Q_stMasterDevState.bDcNotInSync 		:=
	(I_nMasterDevState
		AND 16#1000) = 16#1000;

nMasterDevStatePrev 						:=
	I_nMasterDevState;

// ENDE
END_ACTION

ACTION k_SlaveErrorMessage:
	(* CRC-Fehler ------------------------------------------------------------------------- *)
	(* Anzahl der CRC-Fehler am Port A *)
	IF Q_arrDiagSlaveInfo[nIndexSlave].stPortCRCErrors.portA > 0 THEN
			arrFmEcDiagSlaveError[nIndexErrorMessage] :=
				CONCAT(	'Status EtherCAT-Bus: Teilnehmer: ',
							Q_arrDiagSlaveInfo[nIndexSlave].sName);

			arrFmEcDiagSlaveError[nIndexErrorMessage] :=
				CONCAT(	arrFmEcDiagSlaveError[nIndexErrorMessage],
							', Typ: ');

			arrFmEcDiagSlaveError[nIndexErrorMessage] :=
				CONCAT(	arrFmEcDiagSlaveError[nIndexErrorMessage],
							Q_arrDiagSlaveInfo[nIndexSlave].sType);
	
			arrFmEcDiagSlaveError[nIndexErrorMessage] :=
				CONCAT(	arrFmEcDiagSlaveError[nIndexErrorMessage],
							': Anzahl der CRC-Fehler am Port A: ');

			arrFmEcDiagSlaveError[nIndexErrorMessage] :=
				CONCAT(	arrFmEcDiagSlaveError[nIndexErrorMessage],
							UDINT_TO_STRING(Q_arrDiagSlaveInfo[nIndexSlave].stPortCRCErrors.portA));
	END_IF

	(* Anzahl der CRC-Fehler am Port B *)
	IF Q_arrDiagSlaveInfo[nIndexSlave].stPortCRCErrors.portB > 0 THEN
			arrFmEcDiagSlaveError[nIndexErrorMessage] :=
				CONCAT(	'Status EtherCAT-Bus: Teilnehmer: ',
							Q_arrDiagSlaveInfo[nIndexSlave].sName);

			arrFmEcDiagSlaveError[nIndexErrorMessage] :=
				CONCAT(	arrFmEcDiagSlaveError[nIndexErrorMessage],
							', Typ: ');
	
			arrFmEcDiagSlaveError[nIndexErrorMessage] :=
				CONCAT(	arrFmEcDiagSlaveError[nIndexErrorMessage],
							Q_arrDiagSlaveInfo[nIndexSlave].sType);
	
			arrFmEcDiagSlaveError[nIndexErrorMessage] :=
				CONCAT(	arrFmEcDiagSlaveError[nIndexErrorMessage],
							': Anzahl der CRC-Fehler am Port B: ');
	
			arrFmEcDiagSlaveError[nIndexErrorMessage] :=
				CONCAT(	arrFmEcDiagSlaveError[nIndexErrorMessage],
							UDINT_TO_STRING(Q_arrDiagSlaveInfo[nIndexSlave].stPortCRCErrors.portB));
	END_IF

	(* Anzahl der CRC-Fehler am Port C *)
	IF Q_arrDiagSlaveInfo[nIndexSlave].stPortCRCErrors.portC > 0 THEN
			arrFmEcDiagSlaveError[nIndexErrorMessage] :=
				CONCAT(	'Status EtherCAT-Bus: Teilnehmer: ',
							Q_arrDiagSlaveInfo[nIndexSlave].sName);
	
			arrFmEcDiagSlaveError[nIndexErrorMessage] :=
				CONCAT(	arrFmEcDiagSlaveError[nIndexErrorMessage],
							', Typ: ');

			arrFmEcDiagSlaveError[nIndexErrorMessage] :=
				CONCAT(	arrFmEcDiagSlaveError[nIndexErrorMessage],
							Q_arrDiagSlaveInfo[nIndexSlave].sType);
	
			arrFmEcDiagSlaveError[nIndexErrorMessage] :=
				CONCAT(	arrFmEcDiagSlaveError[nIndexErrorMessage],
							': Anzahl der CRC-Fehler am Port C: ');
	
			arrFmEcDiagSlaveError[nIndexErrorMessage] :=
				CONCAT(	arrFmEcDiagSlaveError[nIndexErrorMessage],
							UDINT_TO_STRING(Q_arrDiagSlaveInfo[nIndexSlave].stPortCRCErrors.portC));
	END_IF
	
	(* Anzahl der CRC-Fehler am Port D *)
	IF Q_arrDiagSlaveInfo[nIndexSlave].stPortCRCErrors.portD > 0 THEN
			arrFmEcDiagSlaveError[nIndexErrorMessage] :=
				CONCAT(	'Status EtherCAT-Bus: Teilnehmer: ',
							Q_arrDiagSlaveInfo[nIndexSlave].sName);
	
			arrFmEcDiagSlaveError[nIndexErrorMessage] :=
				CONCAT(	arrFmEcDiagSlaveError[nIndexErrorMessage],
							', Typ: ');
	
			arrFmEcDiagSlaveError[nIndexErrorMessage] :=
				CONCAT(	arrFmEcDiagSlaveError[nIndexErrorMessage],
							Q_arrDiagSlaveInfo[nIndexSlave].sType);
	
			arrFmEcDiagSlaveError[nIndexErrorMessage] :=
				CONCAT(	arrFmEcDiagSlaveError[nIndexErrorMessage],
							': Anzahl der CRC-Fehler am Port D: ');
	
			arrFmEcDiagSlaveError[nIndexErrorMessage] :=
				CONCAT(	arrFmEcDiagSlaveError[nIndexErrorMessage],
							UDINT_TO_STRING(Q_arrDiagSlaveInfo[nIndexSlave].stPortCRCErrors.portD));
	END_IF
	
	(* ------------------------------------------------------------------------------------ *)
	
	(* Link am angegebenen Port fehlt (Port = A, B, C or D) *)
	IF Q_arrDiagSlaveInfo[nIndexSlave].stState.bMissingLink THEN
	
		arrFmEcDiagSlaveError[nIndexErrorMessage] :=
			CONCAT(	'Fehler EtherCAT-Bus: Teilnehmer: ',
						Q_arrDiagSlaveInfo[nIndexSlave].sName);
	
		arrFmEcDiagSlaveError[nIndexErrorMessage] :=
			CONCAT(	arrFmEcDiagSlaveError[nIndexErrorMessage],
						', Typ: ');
	
		arrFmEcDiagSlaveError[nIndexErrorMessage] :=
			CONCAT(	arrFmEcDiagSlaveError[nIndexErrorMessage],
						Q_arrDiagSlaveInfo[nIndexSlave].sType);
	
		IF Q_arrDiagSlaveInfo[nIndexSlave].stState.bPortA THEN
			arrFmEcDiagSlaveError[nIndexErrorMessage] :=
					CONCAT(	arrFmEcDiagSlaveError[nIndexErrorMessage],
								': Link am Port A fehlt !');
		ELSIF Q_arrDiagSlaveInfo[nIndexSlave].stState.bPortB THEN
			arrFmEcDiagSlaveError[nIndexErrorMessage] :=
				CONCAT(	arrFmEcDiagSlaveError[nIndexErrorMessage],
							': Link am Port B fehlt !');
		ELSIF Q_arrDiagSlaveInfo[nIndexSlave].stState.bPortC THEN
			arrFmEcDiagSlaveError[nIndexErrorMessage] :=
				CONCAT(	arrFmEcDiagSlaveError[nIndexErrorMessage],
							': Link am Port C fehlt !');
		ELSIF Q_arrDiagSlaveInfo[nIndexSlave].stState.bPortD THEN
			arrFmEcDiagSlaveError[nIndexErrorMessage] :=
				CONCAT(	arrFmEcDiagSlaveError[nIndexErrorMessage],
							': Link am Port D fehlt !');
		END_IF
	
		IF nIndexErrorMessage < cMaxAnzahlSlaveError THEN
			nIndexErrorMessage := nIndexErrorMessage + 1;
		ELSE
			RETURN;
		END_IF

	(* Ein zusätzlicher Link wurde am angegebenen Port festgestellt *)
	ELSIF Q_arrDiagSlaveInfo[nIndexSlave].stState.bUnexpectedLink THEN
	
		arrFmEcDiagSlaveError[nIndexErrorMessage] :=
			CONCAT(	'Fehler EtherCAT-Bus: Teilnehmer: ',
						Q_arrDiagSlaveInfo[nIndexSlave].sName);
	
		arrFmEcDiagSlaveError[nIndexErrorMessage] :=
			CONCAT(	arrFmEcDiagSlaveError[nIndexErrorMessage],
						', Typ: ');
	
		arrFmEcDiagSlaveError[nIndexErrorMessage] :=
			CONCAT(	arrFmEcDiagSlaveError[nIndexErrorMessage],
						Q_arrDiagSlaveInfo[nIndexSlave].sType);
	
		IF Q_arrDiagSlaveInfo[nIndexSlave].stState.bPortA THEN
			arrFmEcDiagSlaveError[nIndexErrorMessage] :=
					CONCAT(	arrFmEcDiagSlaveError[nIndexErrorMessage],
								': Ein zusätzlicher Link wurde am Port A festgestellt !');
		ELSIF Q_arrDiagSlaveInfo[nIndexSlave].stState.bPortB THEN
			arrFmEcDiagSlaveError[nIndexErrorMessage] :=
				CONCAT(	arrFmEcDiagSlaveError[nIndexErrorMessage],
								': Ein zusätzlicher Link wurde am Port B festgestellt !');
		ELSIF Q_arrDiagSlaveInfo[nIndexSlave].stState.bPortC THEN
			arrFmEcDiagSlaveError[nIndexErrorMessage] :=
				CONCAT(	arrFmEcDiagSlaveError[nIndexErrorMessage],
								': Ein zusätzlicher Link wurde am Port C festgestellt !');
		ELSIF Q_arrDiagSlaveInfo[nIndexSlave].stState.bPortD THEN
			arrFmEcDiagSlaveError[nIndexErrorMessage] :=
				CONCAT(	arrFmEcDiagSlaveError[nIndexErrorMessage],
								': Ein zusätzlicher Link wurde am Port D festgestellt !');
		END_IF
	
		IF nIndexErrorMessage < cMaxAnzahlSlaveError THEN
			nIndexErrorMessage := nIndexErrorMessage + 1;
		ELSE
			RETURN;
		END_IF

	(* Ein Link ohne Kommunikation wurde festgestellt *)
	ELSIF Q_arrDiagSlaveInfo[nIndexSlave].stState.bLinkError THEN
	
		arrFmEcDiagSlaveError[nIndexErrorMessage] :=
			CONCAT(	'Fehler EtherCAT-Bus: Teilnehmer: ',
						Q_arrDiagSlaveInfo[nIndexSlave].sName);
	
		arrFmEcDiagSlaveError[nIndexErrorMessage] :=
			CONCAT(	arrFmEcDiagSlaveError[nIndexErrorMessage],
						', Typ: ');
	
		arrFmEcDiagSlaveError[nIndexErrorMessage] :=
			CONCAT(	arrFmEcDiagSlaveError[nIndexErrorMessage],
						Q_arrDiagSlaveInfo[nIndexSlave].sType);
	
		IF Q_arrDiagSlaveInfo[nIndexSlave].stState.bPortA THEN
			arrFmEcDiagSlaveError[nIndexErrorMessage] :=
					CONCAT(	arrFmEcDiagSlaveError[nIndexErrorMessage],
								': Am Port A wurde ein Link ohne Kommunikation festgestellt !');
		ELSIF Q_arrDiagSlaveInfo[nIndexSlave].stState.bPortB THEN
			arrFmEcDiagSlaveError[nIndexErrorMessage] :=
				CONCAT(	arrFmEcDiagSlaveError[nIndexErrorMessage],
								': Am Port B wurde ein Link ohne Kommunikation festgestellt !');
		ELSIF Q_arrDiagSlaveInfo[nIndexSlave].stState.bPortC THEN
			arrFmEcDiagSlaveError[nIndexErrorMessage] :=
				CONCAT(	arrFmEcDiagSlaveError[nIndexErrorMessage],
								': Am Port C wurde ein Link ohne Kommunikation festgestellt !');
		ELSIF Q_arrDiagSlaveInfo[nIndexSlave].stState.bPortD THEN
			arrFmEcDiagSlaveError[nIndexErrorMessage] :=
				CONCAT(	arrFmEcDiagSlaveError[nIndexErrorMessage],
								': Am Port D wurde ein Link ohne Kommunikation festgestellt !');
		END_IF
	
		IF nIndexErrorMessage < cMaxAnzahlSlaveError THEN
			nIndexErrorMessage := nIndexErrorMessage + 1;
		ELSE
			RETURN;
		END_IF
	
	END_IF

	
	(* Fehler Slave nicht erkannt *)
	IF Q_arrDiagSlaveInfo[nIndexSlave].stState.bNoCommToSlave THEN
	
		arrFmEcDiagSlaveError[nIndexErrorMessage] :=
			CONCAT(	'Fehler EtherCAT-Bus: Teilnehmer: ',
						Q_arrDiagSlaveInfo[nIndexSlave].sName);
	
		arrFmEcDiagSlaveError[nIndexErrorMessage] :=
			CONCAT(	arrFmEcDiagSlaveError[nIndexErrorMessage],
						', Typ: ');
	
		arrFmEcDiagSlaveError[nIndexErrorMessage] :=
			CONCAT(	arrFmEcDiagSlaveError[nIndexErrorMessage],
						Q_arrDiagSlaveInfo[nIndexSlave].sType);

		arrFmEcDiagSlaveError[nIndexErrorMessage] :=
			CONCAT(	arrFmEcDiagSlaveError[nIndexErrorMessage],
						': State: ');
	
		CASE Q_arrDiagSlaveInfo[nIndexSlave].stState.eEcState OF
	
		eEcState_UNDEFINED:	arrFmEcDiagSlaveError[nIndexErrorMessage] :=
										CONCAT(	arrFmEcDiagSlaveError[nIndexErrorMessage],
													'UNDEFINED');
		eEcState_INIT:			arrFmEcDiagSlaveError[nIndexErrorMessage] :=
										CONCAT(	arrFmEcDiagSlaveError[nIndexErrorMessage],
													'INIT / NO COMMUNICATION');
		eEcState_PREOP:		arrFmEcDiagSlaveError[nIndexErrorMessage] :=
										CONCAT(	arrFmEcDiagSlaveError[nIndexErrorMessage],
													'PREOP');
		eEcState_BOOT:			arrFmEcDiagSlaveError[nIndexErrorMessage] :=
										CONCAT(	arrFmEcDiagSlaveError[nIndexErrorMessage],
													'BOOT');
		eEcState_SAFEOP:		arrFmEcDiagSlaveError[nIndexErrorMessage] :=
										CONCAT(	arrFmEcDiagSlaveError[nIndexErrorMessage],
													'SAFEOP');
		eEcState_OP:			arrFmEcDiagSlaveError[nIndexErrorMessage] :=
										CONCAT(	arrFmEcDiagSlaveError[nIndexErrorMessage],
													'OP');
		END_CASE
	
		IF nIndexErrorMessage < cMaxAnzahlSlaveError THEN
			nIndexErrorMessage := nIndexErrorMessage + 1;
		ELSE
			RETURN;
		END_IF
	END_IF
	
	(* B E *)
END_ACTION

END_FUNCTION_BLOCK

// POUs/EtherCATDiagnose/FB_EtherCATFrameDiag
FUNCTION_BLOCK FB_EtherCATFrameDiag
VAR_INPUT
	I_nFrameXWcState 		: WORD;
	I_nFrameState			: WORD;
END_VAR
VAR_OUTPUT
	Q_bFrameWcStateOK		: BOOL;
	Q_bFrameStateOK		: BOOL;
END_VAR

// set/clear frame flag
Q_bFrameWcStateOK := ((I_nFrameXWcState AND 16#FFFF) = 0);

Q_bFrameStateOK	:= ((I_nFrameState AND 16#FFFF) = 0);

END_FUNCTION_BLOCK

// POUs/EtherCATDiagnose/FB_IoLinkFehler
(*
Date				| Version		| created under			| Author				| Remark 
---------------------------------------------------------------------------------------- 
03/10/2017		| 1.0.0			| V2.11.2258				| H.Gennet			| first release 
*)
(*Pro Zyklus nur einen der 4 Channels, nacheinander.*)
FUNCTION_BLOCK FB_IoLinkFehler
VAR
	// Baustein zum Zusammenfügen von Texten in ein String
	fbFormat 	: Tc2_Utilities.FB_FormatString;

	// Zähler
	nCounter 	: INT; 				(*Zähler für das nState Array*)
	nChannel		: INT;				(*Zähler + 1*)

	// Zwischenspeicher der Input Stati zur besseren Auswertung
	nState 		: ARRAY [0..3] OF USINT;
	
	arrLetzteFehlermeldung	: ARRAY [0..3] OF Tc2_System.T_MaxString;
	arrVerzMeld					: ARRAY [0..3] OF TON;

END_VAR
VAR_IN_OUT
	IQ_stMeldung	: ST_MeldIOLinkKlemme;
END_VAR

VAR_INPUT
	(*BMK Input händisch als String*)
	I_sBMK : 	Tc2_System.T_MaxString;

	(*Input der einzelnen Stati*)
	I_nStateCh1	: USINT;
	I_nStateCh2	: USINT;
	I_nStateCh3	: USINT;
	I_nStateCh4	: USINT;
END_VAR

VAR_OUTPUT
	Q_arrFehlermeldung : ARRAY [0..3] OF Tc2_System.T_MaxString;	// Output der Fehlermeldungen als String-Array
END_VAR

(*Übertragung der einzelnen Stati in ein Array*)
nState[0] := I_nStateCh1;
nState[1] := I_nStateCh2;
nState[2] := I_nStateCh3;
nState[3] := I_nStateCh4;

(*Zurücksetzen des Counters, wenn dieser größer als 3 ist*)
IF nCounter > 3 THEN
	nCounter := 0;
END_IF

nChannel := nCounter +1;
(*Abfrage der aktuellen Stati*)
CASE nState[nCounter] OF
	(*16#00:
		(*Port diasbled*)
		fbFormat(sFormat := '%s Ch %d: Kein Teilnehmer an Ch %d  angeschlossen!',arg1:=F_STRING(sBMK), arg2:=F_INT(nChannel), sOut => sFehlermeldung[nCounter]);
	16#01:
		(*Port in std dig in*)
		fbFormat(sFormat := '%s Ch %d: ist als Standard Input definiert!',arg1:=F_STRING(sBMK), arg2:=F_INT(nChannel), sOut => sFehlermeldung[nCounter]);
	16#02:
		(*Port in std dig out*)
		fbFormat(sFormat := '%s Ch %d: ist als Standard Output definiert!',arg1:=F_STRING(sBMK), arg2:=F_INT(nChannel), sOut => sFehlermeldung[nCounter]);
	16#03:
		(*Port in communikation OP*)
		fbFormat(sFormat := '%s Ch %d: befindet sich im Status OP!',arg1:=F_STRING(sBMK), arg2:=F_INT(nChannel), sOut => sFehlermeldung[nCounter]);*)
	16#04:
		(*Port in communikation Comport*)
		fbFormat(sFormat := '%s Ch %d: Port in communikation Comport!',arg1:=F_STRING(I_sBMK), arg2:=F_INT(nChannel), sOut => Q_arrFehlermeldung[nCounter]);
	16#0B:
		(*Teilnehmer befindet sich im Teach-in Modus*)
		fbFormat(sFormat := '%s Ch %d: eingeteacht!',arg1:=F_STRING(I_sBMK), arg2:=F_INT(nChannel), sOut => Q_arrFehlermeldung[nCounter]);
	16#10:
		(*Watchdog detected*)
		fbFormat(sFormat := '%s Ch %d: Watchdog hat ausgelöst!',arg1:=F_STRING(I_sBMK), arg2:=F_INT(nChannel), sOut => Q_arrFehlermeldung[nCounter]);
	16#20:
		(*internal Error*)
		fbFormat(sFormat := '%s Ch %d: Es gibt einen internen Fehler!',arg1:=F_STRING(I_sBMK), arg2:=F_INT(nChannel), sOut => Q_arrFehlermeldung[nCounter]);
	16#30,16#B0: (*Bei einer falschen Device ID (DeviceDescription) springt der Status zwischen 16#30 und 16#B0*)
		(*invalid Device ID*)
		fbFormat(sFormat := '%s Ch %d: Die Device ID ist fehlerhaft!',arg1:=F_STRING(I_sBMK), arg2:=F_INT(nChannel), sOut => Q_arrFehlermeldung[nCounter]); (* Bitte die korrekte Device Describtion einlesen und den korrekten Teilnehmer auswählen*)
	16#40:
		(*invalid Vendor ID*)
		fbFormat(sFormat := '%s Ch %d: Die Vendor ID ist fehlerhaft!',arg1:=F_STRING(I_sBMK), arg2:=F_INT(nChannel), sOut => Q_arrFehlermeldung[nCounter]);	(* Bitte in der Device Describtion korrigieren. Die Vendor IDs können über Io-Link.com abgerufen werden *)
	16#50:
		(*invalid IO-Link Error*)
		fbFormat(sFormat := '%s Ch %d: Es liegt ein IO-Link Error vor!',arg1:=F_STRING(I_sBMK), arg2:=F_INT(nChannel), sOut => Q_arrFehlermeldung[nCounter]);
	16#60:
		(*invalid Frame Capability*)
		fbFormat(sFormat := '%s Ch %d: Der aktuelle Frame ist ungültig!',arg1:=F_STRING(I_sBMK), arg2:=F_INT(nChannel), sOut => Q_arrFehlermeldung[nCounter]);
	16#70:
		(*invalid Cycle Time*)
		fbFormat(sFormat := '%s Ch %d: Die Zylkuszeit ist ungültig. Bitte die Einstellungen überprüfen!',arg1:=F_STRING(I_sBMK), arg2:=F_INT(nChannel), sOut => Q_arrFehlermeldung[nCounter]);
	16#80:
		(*invalid PD in length*)
		fbFormat(sFormat := '%s Ch %d: Die Länge der eingehenden Prozessdaten passt nicht mit der erwarteten Länge zusammen!',arg1:=F_STRING(I_sBMK), arg2:=F_INT(nChannel), sOut => Q_arrFehlermeldung[nCounter]);
	16#90:
		(*invalid PD out length*)
		fbFormat(sFormat := '%s Ch %d: Die Länge der ausgehenden Prozessdaten passt nicht mit der erwarteten Länge zusammen!',arg1:=F_STRING(I_sBMK), arg2:=F_INT(nChannel), sOut => Q_arrFehlermeldung[nCounter]);
	16#A0:
		(*no Device detected*)
		fbFormat(sFormat := '%s Ch %d: Der Teilnehmer hat den Kontakt verloren!',arg1:=F_STRING(I_sBMK), arg2:=F_INT(nChannel), sOut => Q_arrFehlermeldung[nCounter]); (* Bitte die Anschlüsse und Verbindungskabel prüfen. Wenn dort nichts vorliegt kann der Teilnehmer defekt sein*)
	ELSE
		IF (nState[nCounter] > 16#03) THEN
			(*Unbekannter Zustand, der nicht im Infosys definiert ist*)
			fbFormat(sFormat := '%s Ch %d: Unbekannter Status!',arg1:=F_STRING(I_sBMK), arg2:=F_INT(nChannel), sOut => Q_arrFehlermeldung[nCounter]);
		ELSE
			Q_arrFehlermeldung[nCounter] := '';
		END_IF
END_CASE

nCounter := nCounter+1;

// Zuweisung der Meldungen
IQ_stMeldung.SourceName	:= I_sBMK;

arrVerzMeld[0](
	IN := Q_arrFehlermeldung[0] <> ''
				AND Q_arrFehlermeldung[0] = arrLetzteFehlermeldung[0],
	PT := t#500MS
);

arrVerzMeld[1](
	IN := Q_arrFehlermeldung[1] <> ''
				AND Q_arrFehlermeldung[1] = arrLetzteFehlermeldung[1],
	PT := t#500MS
);

arrVerzMeld[2](
	IN := Q_arrFehlermeldung[2] <> ''
				AND Q_arrFehlermeldung[2] = arrLetzteFehlermeldung[2],
	PT := t#500MS
);

arrVerzMeld[3](
	IN := Q_arrFehlermeldung[3] <> ''
				AND Q_arrFehlermeldung[3] = arrLetzteFehlermeldung[3],
	PT := t#500MS
);

IQ_stMeldung.bMeld1	:= arrVerzMeld[0].Q;
IQ_stMeldung.bMeld2	:= arrVerzMeld[1].Q;
IQ_stMeldung.bMeld3	:= arrVerzMeld[2].Q;
IQ_stMeldung.bMeld4	:= arrVerzMeld[3].Q;
IQ_stMeldung.sText1	:= Q_arrFehlermeldung[0];
IQ_stMeldung.sText2	:= Q_arrFehlermeldung[1];
IQ_stMeldung.sText3	:= Q_arrFehlermeldung[2];
IQ_stMeldung.sText4	:= Q_arrFehlermeldung[3];


arrLetzteFehlermeldung[0] :=  Q_arrFehlermeldung[0];
arrLetzteFehlermeldung[1] :=  Q_arrFehlermeldung[1];
arrLetzteFehlermeldung[2] :=  Q_arrFehlermeldung[2];
arrLetzteFehlermeldung[3] :=  Q_arrFehlermeldung[3];

// ENDE

END_FUNCTION_BLOCK

// POUs/Grundstellung/FB_UniGrdstlgAbl
// Dieser Grundstellungsablauf besteht aus einer Schrittkette mit insgesamt 9 einzelnen Schritten.
// Gesteuert wird er über zwei HMI-Schnittstellen und weiteren Eingängen zum Starten der Grundstellung
FUNCTION_BLOCK FB_UniGrdstlgAbl
VAR_INPUT

	I_sStatName			:Tc2_System.T_MaxString;	// Aktueller Stationsname für Fehlermeldungen

	I_bHandbetrAktiv	:BOOL;	// Betriebsart, Schutzbereich etc.
	I_bGrdstAnwahlFrg	:BOOL;	// Betriebsart, Schutzbereich etc.

	I_bLoeschDatenPos :BOOL;	// Grundstellungsablauf-Anwahl durch Datensatz löschen in der Teileverfolgung
	I_bGrdstlgAnwTast :BOOL;	// Grundstellungsablauf-Anwahl durch Paneltaste, Softkey etc.
	I_bGrdstlgAnfStat	:BOOL;	// Grundstellungsablauf-Anwahl durch extern z.B. Referenzablauf. Bei fallender Flanke wird die Grundstellung wieder abgewählt, bzw. umgeschaltet
	
	I_bDatenVorh		:BOOL;	// Sind Daten vorhanden wird das Lösch-Bit gesetzt
	I_bSensPosFreiErk	:BOOL:= TRUE;	// Optional: Erkennung Teileentnahme. Grundstellung ist erst zuende, wenn dieses Bit TRUE ist.
	I_bTeileEntnahmeNoetig	: BOOL;	// Nur für eine Melden, dass nach der erfolgreichen Grundstellungsfahrt das Teil entnommen werden soll. Die Meldung bleibt so lange an wie die Grundstellung aktiv ist oder dieses Bit gesetzt
	 
	I_bGrdstStep1End	:BOOL:= TRUE;	// Rückmeldung Schritt 1 fertig
	I_bGrdstStep2End	:BOOL:= TRUE;	// Rückmeldung Schritt 2 fertig
	I_bGrdstStep3End	:BOOL:= TRUE;	// Rückmeldung Schritt 3 fertig
	I_bGrdstStep4End	:BOOL:= TRUE;	// Rückmeldung Schritt 4 fertig
	I_bGrdstStep5End	:BOOL:= TRUE;	// Rückmeldung Schritt 5 fertig
	I_bGrdstStep6End	:BOOL:= TRUE;	// Rückmeldung Schritt 6 fertig
	I_bGrdstStep7End	:BOOL:= TRUE;	// Rückmeldung Schritt 7 fertig
	I_bGrdstStep8End	:BOOL:= TRUE;	// Rückmeldung Schritt 8 fertig
	I_bGrdstStep9End	:BOOL:= TRUE;	// Rückmeldung Schritt 9 fertig

	I_bParamEinzelschritte	: BOOL;	// Wenn dieser Parameter an ist, dann sind die Schritte nur einzeln an. Also wenn Q_bGrdstStep2Akt an geht, geht Q_bGrdstStep1Akt aus.
END_VAR
VAR_IN_OUT

	IQ_stUniAnstgEinzelHMI	:ST_UniGrdstlgAbl;	// HMI-Struktur Einzelposition
	IQ_stUniAnstgGesamtHMI	:ST_UniGrdstlgAbl;	// HMI-Struktur Anlagenbereich/Gesamtanlage, Liste mit allen Grundstellungsabläufen

END_VAR
VAR_OUTPUT

	Q_bGrdstAblAktiv	:BOOL;	// Gesamtablauf Aktiv
	Q_bGrdstAblReset	:BOOL;	// Gesamtablauf 1x Reset
	Q_bGrdstAblEnde	:BOOL;	// Gesamtablauf Ausgeführt
	
	Q_bDatenLoeschen	:BOOL;	// Ein vorhandener Datensatz soll gelöscht werden
	 
	Q_bGrdstStep1Akt	:BOOL;	// Ist TRUE sobald die Grundstellung aktiv ist. Wenn der Parameter I_bParamEinzelschritte aktiv ist, dann wirds FALSE wenn der nächste Schritt aktiv ist.
	Q_bGrdstStep2Akt	:BOOL;	// Ist TRUE sobald die Weiterschaltbedingung vom vorherigen TRUE ist. Wenn der Parameter I_bParamEinzelschritte aktiv ist, dann wirds FALSE wenn der nächste Schritt aktiv ist.
	Q_bGrdstStep3Akt	:BOOL;	// Ist TRUE sobald die Weiterschaltbedingung vom vorherigen TRUE ist. Wenn der Parameter I_bParamEinzelschritte aktiv ist, dann wirds FALSE wenn der nächste Schritt aktiv ist.
	Q_bGrdstStep4Akt	:BOOL;	// Ist TRUE sobald die Weiterschaltbedingung vom vorherigen TRUE ist. Wenn der Parameter I_bParamEinzelschritte aktiv ist, dann wirds FALSE wenn der nächste Schritt aktiv ist.
	Q_bGrdstStep5Akt	:BOOL;	// Ist TRUE sobald die Weiterschaltbedingung vom vorherigen TRUE ist. Wenn der Parameter I_bParamEinzelschritte aktiv ist, dann wirds FALSE wenn der nächste Schritt aktiv ist.
	Q_bGrdstStep6Akt	:BOOL;	// Ist TRUE sobald die Weiterschaltbedingung vom vorherigen TRUE ist. Wenn der Parameter I_bParamEinzelschritte aktiv ist, dann wirds FALSE wenn der nächste Schritt aktiv ist.
	Q_bGrdstStep7Akt	:BOOL;	// Ist TRUE sobald die Weiterschaltbedingung vom vorherigen TRUE ist. Wenn der Parameter I_bParamEinzelschritte aktiv ist, dann wirds FALSE wenn der nächste Schritt aktiv ist.
	Q_bGrdstStep8Akt	:BOOL;	// Ist TRUE sobald die Weiterschaltbedingung vom vorherigen TRUE ist. Wenn der Parameter I_bParamEinzelschritte aktiv ist, dann wirds FALSE wenn der nächste Schritt aktiv ist.
	Q_bGrdstStep9Akt	:BOOL;	// Ist TRUE sobald die Weiterschaltbedingung vom vorherigen TRUE ist. Dieser Schritt bleibt solange TRUE wie die Grundstellung aktiv ist.

	Q_bGrdstlgMeldg	:BOOL;	// Grundstellung-Meldung für Paneltaste, Softkey etc. mit Blinktakt wenn aktiv. Durchgehen TRUE, wenn Grundstellung Ende
END_VAR
VAR

	rtrigImpAnAbw		:R_TRIG;
	rtrigDatenLoeschen:R_TRIG;
	bGrdst1xAngw		:BOOL;

	nStepState			:INT;
END_VAR

	(*Uni.- Grundstellungsablauf*)
	
	(**************************************************)	
	(*Grundstellung An.-Abwahl*)

	a_AnAbwahl();
	
	(**************************************************)	
	(*Grundstellung Step-Ablauf*)

	b_StepAblauf();

	(**************************************************)	
	(*Zustände anzeigen*)

	y_ZustAnzg();

	(**************************************************)	
	(*Meldungen ausgeben*)

	z_HinwMeld();
	
	(**************************************************)

ACTION a_AnAbwahl:
	
//****************************************************************************************************
// Grundstellung An.-Abwahl
	
	rtrigDatenLoeschen(CLK:= I_bLoeschDatenPos);
									  
	rtrigImpAnAbw (CLK:= (IQ_stUniAnstgEinzelHMI.stHandFktHMI[1].bySwitch > 0
								OR IQ_stUniAnstgGesamtHMI.stHandFktHMI[1].bySwitch > 0
								OR I_bGrdstlgAnwTast
								OR (I_bGrdstlgAnfStat
									 AND NOT bGrdst1xAngw) 
								OR (NOT I_bGrdstlgAnfStat
									 AND bGrdst1xAngw))
								AND (I_bGrdstAnwahlFrg
									 AND I_bHandbetrAktiv));

//****************************************************************************************************
//ToDo teilweise nur Anwahl /direkter zugriff auf Teileverfolgung...

	Q_bGrdstAblReset:= FALSE;
	
	IF NOT I_bHandbetrAktiv
		THEN
			Q_bGrdstAblAktiv:= FALSE;
			bGrdst1xAngw	 := FALSE;	
			nStepState		 := 0;			
	ELSIF rtrigImpAnAbw.Q
		THEN
			Q_bGrdstAblAktiv:= NOT Q_bGrdstAblAktiv;
			Q_bGrdstAblReset:= Q_bGrdstAblAktiv;
			bGrdst1xAngw	 := I_bGrdstlgAnfStat; //ToDo
			nStepState		 := 0;
			
	ELSIF rtrigDatenLoeschen.Q
		OR (I_bLoeschDatenPos
			AND NOT Q_bGrdstAblAktiv)
		THEN
			Q_bGrdstAblAktiv	:= TRUE;
			Q_bGrdstAblReset:= Q_bGrdstAblAktiv;
			nStepState		 := 0;
	END_IF

//****************************************************************************************************
//
END_ACTION

ACTION b_StepAblauf:
	
//****************************************************************************************************
// Grundstellung Step-Ablauf

	CASE nStepState OF
0:	//Initialisierung

	Q_bDatenLoeschen:=	
	Q_bGrdstStep1Akt:=
	Q_bGrdstStep2Akt:=
	Q_bGrdstStep3Akt:=
	Q_bGrdstStep4Akt:=
	Q_bGrdstStep5Akt:=
	Q_bGrdstStep6Akt:=
	Q_bGrdstStep7Akt:=
	Q_bGrdstStep8Akt:=
	Q_bGrdstStep9Akt:= FALSE;

	IF Q_bGrdstAblAktiv THEN
		nStepState:= 1;
	END_IF
	
1:	//Ablauf Step 1
	Q_bGrdstStep1Akt:= TRUE;
	
	IF I_bGrdstStep1End THEN
		nStepState:= 2;
		Q_bGrdstStep1Akt	:= NOT I_bParamEinzelschritte;
	END_IF
	
2:	//Ablauf Step 2
	Q_bGrdstStep2Akt:= TRUE;
	
	IF I_bGrdstStep2End THEN
		nStepState:= 3;
		Q_bGrdstStep2Akt	:= NOT I_bParamEinzelschritte;
	END_IF
	
3:	//Ablauf Step 3
	Q_bGrdstStep3Akt:= TRUE;
	
	IF I_bGrdstStep3End THEN
		nStepState:= 4;
		Q_bGrdstStep3Akt	:= NOT I_bParamEinzelschritte;
	END_IF
	
4:	//Ablauf Step 4
	Q_bGrdstStep4Akt:= TRUE;
	
	IF I_bGrdstStep4End THEN
		nStepState:= 5;
		Q_bGrdstStep4Akt	:= NOT I_bParamEinzelschritte;
	END_IF
	
5:	//Ablauf Step 5
	Q_bGrdstStep5Akt:= TRUE;
	
	IF I_bGrdstStep5End THEN
		nStepState:= 6;
		Q_bGrdstStep5Akt	:= NOT I_bParamEinzelschritte;
	END_IF
	
6:	//Ablauf Step 6
	Q_bGrdstStep6Akt:= TRUE;
	
	IF I_bGrdstStep6End THEN
		nStepState:= 7;
		Q_bGrdstStep6Akt	:= NOT I_bParamEinzelschritte;
	END_IF
	
7:	//Ablauf Step 7
	Q_bGrdstStep7Akt:= TRUE;
	
	IF I_bGrdstStep7End THEN
		nStepState:= 8;
		Q_bGrdstStep7Akt	:= NOT I_bParamEinzelschritte;
	END_IF
	
8:	//Ablauf Step 8
	Q_bGrdstStep8Akt:= TRUE;
	
	IF I_bGrdstStep8End THEN
		nStepState:= 9;
		Q_bGrdstStep8Akt	:= NOT I_bParamEinzelschritte;
	END_IF
	
9:	//Ablauf Step 9
	Q_bGrdstStep9Akt:= TRUE;
	
	IF I_bGrdstStep9End THEN
		nStepState:= 10;
	END_IF
	
10://Datenabfrage, wenn Daten zum löschen vorhanden sind, bleibt das Lösch-Bit an
	
	IF I_bDatenVorh
		THEN
			Q_bDatenLoeschen	:= TRUE;	
		ELSE
			Q_bDatenLoeschen	:= FALSE;
			nStepState:= 99;
   END_IF

99://Ablaufende	

	END_CASE	

//****************************************************************************************************

	Q_bGrdstAblEnde:= nStepState = 99
							AND I_bSensPosFreiErk;
 
//****************************************************************************************************
END_ACTION

ACTION y_ZustAnzg:

//****************************************************************************************************
// Zustände anzeigen

	IF I_bGrdstAnwahlFrg
		AND I_bHandbetrAktiv
	THEN	// Funktion freigegeben
			IQ_stUniAnstgEinzelHMI.stHandFktHMI[1].sColour	:= cDefaultAsString;
			IQ_stUniAnstgEinzelHMI.stHandFktHMI[1].sText		:= 'ausführen';
			IQ_stUniAnstgGesamtHMI.stHandFktHMI[1].sColour	:= cDefaultAsString;
			IQ_stUniAnstgGesamtHMI.stHandFktHMI[1].sText		:= 'ausführen';
			IQ_stUniAnstgEinzelHMI.stHandFktHMI[1].byStatus	:= 0;
			IQ_stUniAnstgGesamtHMI.stHandFktHMI[1].byStatus	:= 0;
			IQ_stUniAnstgEinzelHMI.stHandFktHMI[1].iDisplayMode	:= 0;
			IQ_stUniAnstgGesamtHMI.stHandFktHMI[1].iDisplayMode	:= 0;

		IF Q_bGrdstAblAktiv
			AND NOT Q_bGrdstAblEnde
		THEN	// Handfunktion aktiv
			IQ_stUniAnstgEinzelHMI.stHandFktHMI[1].sColour	:= cGelbAsString;
			IQ_stUniAnstgEinzelHMI.stHandFktHMI[1].sText		:= 'ausführen';
			IQ_stUniAnstgGesamtHMI.stHandFktHMI[1].sColour	:= cGelbAsString;
			IQ_stUniAnstgGesamtHMI.stHandFktHMI[1].sText		:= 'ausführen';
			IQ_stUniAnstgEinzelHMI.stHandFktHMI[1].byStatus	:= 0;
			IQ_stUniAnstgGesamtHMI.stHandFktHMI[1].byStatus	:= 0;
			IQ_stUniAnstgEinzelHMI.stHandFktHMI[1].iDisplayMode	:= 2;
			IQ_stUniAnstgGesamtHMI.stHandFktHMI[1].iDisplayMode	:= 2;
		END_IF
		
		IF Q_bGrdstAblEnde
		THEN	// Handfunktion ausgeführt
			IQ_stUniAnstgEinzelHMI.stHandFktHMI[1].sColour:= cGruenAsString;
			IQ_stUniAnstgEinzelHMI.stHandFktHMI[1].sText:= 'ausgeführt';
			IQ_stUniAnstgGesamtHMI.stHandFktHMI[1].sColour:= cGruenAsString;
			IQ_stUniAnstgGesamtHMI.stHandFktHMI[1].sText:= 'ausgeführt';
			IQ_stUniAnstgEinzelHMI.stHandFktHMI[1].byStatus:= 0;
			IQ_stUniAnstgGesamtHMI.stHandFktHMI[1].byStatus:= 0;
			IQ_stUniAnstgEinzelHMI.stHandFktHMI[1].iDisplayMode	:= 0;
			IQ_stUniAnstgGesamtHMI.stHandFktHMI[1].iDisplayMode	:= 0;
		END_IF
		
	ELSE	// Funktion gesperrt
		IQ_stUniAnstgEinzelHMI.stHandFktHMI[1].sColour	:= cDefaultAsString;
		IQ_stUniAnstgEinzelHMI.stHandFktHMI[1].sText		:= 'ausführen';
		IQ_stUniAnstgGesamtHMI.stHandFktHMI[1].sColour	:= cDefaultAsString;
		IQ_stUniAnstgGesamtHMI.stHandFktHMI[1].sText		:= 'ausführen';
		IQ_stUniAnstgEinzelHMI.stHandFktHMI[1].byStatus	:= 1;
		IQ_stUniAnstgGesamtHMI.stHandFktHMI[1].byStatus	:= 1;
		IQ_stUniAnstgEinzelHMI.stHandFktHMI[1].iDisplayMode	:= 0;
		IQ_stUniAnstgGesamtHMI.stHandFktHMI[1].iDisplayMode	:= 0;
	END_IF
END_ACTION

ACTION z_HinwMeld:

//****************************************************************************************************
// Fehler-Meldungen ausgeben

	IQ_stUniAnstgEinzelHMI.stMeldAusgHMI.SourceID		:= 0;	// Nicht mehr verwendet
	IQ_stUniAnstgEinzelHMI.stMeldAusgHMI.SourceName		:= I_sStatName;

	IF bTestMeldGrdstlg
	THEN
		IQ_stUniAnstgEinzelHMI.stMeldAusgHMI.bMeldAktiv						:=
		IQ_stUniAnstgEinzelHMI.stMeldAusgHMI.bMeldDonemitEntnahme		:= 
		IQ_stUniAnstgEinzelHMI.stMeldAusgHMI.bMeldDoneOhneEntnahme		:= TRUE;
	ELSIF nStepState >= 1 THEN
		IQ_stUniAnstgEinzelHMI.stMeldAusgHMI.bMeldAktiv					:= TRUE; 
		IQ_stUniAnstgEinzelHMI.stMeldAusgHMI.bMeldDonemitEntnahme	:= FALSE;
		IQ_stUniAnstgEinzelHMI.stMeldAusgHMI.bMeldDoneOhneEntnahme	:= FALSE;
		IF nStepState >= 10 THEN
			IQ_stUniAnstgEinzelHMI.stMeldAusgHMI.bMeldAktiv			:= FALSE;
			IF I_bTeileEntnahmeNoetig
			THEN 
				IQ_stUniAnstgEinzelHMI.stMeldAusgHMI.bMeldDonemitEntnahme	:= TRUE;
			ELSE 
				IQ_stUniAnstgEinzelHMI.stMeldAusgHMI.bMeldDoneOhneEntnahme	:= TRUE;
			END_IF
		END_IF
	ELSE
		IQ_stUniAnstgEinzelHMI.stMeldAusgHMI.bMeldAktiv						:=
		IQ_stUniAnstgEinzelHMI.stMeldAusgHMI.bMeldDonemitEntnahme		:= 
		IQ_stUniAnstgEinzelHMI.stMeldAusgHMI.bMeldDoneOhneEntnahme		:= FALSE;
   END_IF
	
//****************************************************************************************************
// Hardware-Meldungen

	Q_bGrdstlgMeldg:= (Q_bGrdstAblAktiv AND bTaktLangsam) OR	Q_bGrdstAblEnde;
	
//****************************************************************************************************
END_ACTION

END_FUNCTION_BLOCK

// POUs/Grundstellung/FB_UniGrdstlgAblBereich
// Dieser Grundstellungsablauf hat noch einen zusätzlichen Ein-Ausgang für einen Grundstellungsbereich (z.B. einen Schutzbereich)
// Das Ganze verhält sich aber so, dass die VAR_IN_OUT für Bereich von allen Grundstellungsabläufen beschrieben wird, an die diese Struktur angelegt wird.
// Somit wird nur der Zustand vom letzten Grundstellungsablauf, an dem diese Struktur angelegt sind, angezeigt.
// hat aber sonst die gleiche Funktion wie der FB_UniGrdstlgAbl
FUNCTION_BLOCK FB_UniGrdstlgAblBereich
VAR_INPUT

	I_sStatName			:Tc2_System.T_MaxString;	// Aktueller Stationsname für Fehlermeldungen

	I_bHandbetrAktiv	:BOOL;	//	Betriebsart, Schutzbereich etc.
	I_bGrdstAnwahlFrg	:BOOL;	// Betriebsart, Schutzbereich etc.
	
	I_bLoeschDatenPos :BOOL;	// Grundstellungsablauf-Anwahl durch Datensatz löschen in der Teileverfolgung
	I_bGrdstlgAnwTast :BOOL;	// Grundstellungsablauf-Anwahl durch Paneltaste, Softkey etc.
	I_bGrdstlgAnfStat	:BOOL;	// Grundstellungsablauf-Anwahl durch extern z.B. Referenzablauf. Bei fallender Flanke wird die Grundstellung wieder abgewählt, bzw. umgeschaltet

	I_bDatenVorh		:BOOL;	// Sind Daten vorhanden wird das Lösch-Bit gesetzt
	I_bSensPosFreiErk	:BOOL:= TRUE;	// Optional: Erkennung Teileentnahme. Grundstellung ist erst zuende, wenn dieses Bit TRUE ist.
	I_bTeileEntnahmeNoetig	: BOOL;	// Nur für eine Melden, dass nach der erfolgreichen Grundstellungsfahrt das Teil entnommen werden soll. Die Meldung bleibt so lange an wie die Grundstellung aktiv ist oder dieses Bit gesetzt
	 
	I_bGrdstStep1End	:BOOL:= TRUE;	// Rückmeldung Schritt 1 fertig
	I_bGrdstStep2End	:BOOL:= TRUE;	// Rückmeldung Schritt 2 fertig
	I_bGrdstStep3End	:BOOL:= TRUE;	// Rückmeldung Schritt 3 fertig
	I_bGrdstStep4End	:BOOL:= TRUE;	// Rückmeldung Schritt 4 fertig
	I_bGrdstStep5End	:BOOL:= TRUE;	// Rückmeldung Schritt 5 fertig
	I_bGrdstStep6End	:BOOL:= TRUE;	// Rückmeldung Schritt 6 fertig
	I_bGrdstStep7End	:BOOL:= TRUE;	// Rückmeldung Schritt 7 fertig
	I_bGrdstStep8End	:BOOL:= TRUE;	// Rückmeldung Schritt 8 fertig
	I_bGrdstStep9End	:BOOL:= TRUE;	// Rückmeldung Schritt 9 fertig

	I_bParamEinzelschritte	: BOOL;	// Wenn dieser Parameter an ist, dann sind die Schritte nur einzeln an. Also wenn Q_bGrdstStep2Akt an geht, geht Q_bGrdstStep1Akt aus.
END_VAR
VAR_IN_OUT
	IQ_stUniAnstgEinzelHMI	:ST_UniGrdstlgAbl;	//HMI-Struktur Einzelposition
	IQ_stUniAnstgBereichHMI	:ST_UniGrdstlgAbl;	//HMI-Struktur für einen Bereich, z.B. Schutzbereich. Über diese Schnittstelle ist nur einschalten möglich, nicht ausschalten. Es wird nur der Zustand von dem letzten Grundstellungsablauf mit dieser Schnittstelle angezeigt.
	IQ_stUniAnstgGesamtHMI	:ST_UniGrdstlgAbl;	//HMI-Struktur Anlagenbereich/Gesamtanlage, Liste mit allen Grundstellungsabläufen
END_VAR
VAR_OUTPUT
	Q_bGrdstAblAktiv	:BOOL;	//Grundstellungsablauf Aktiv
	Q_bGrdstAblReset	:BOOL;	//Grundstellungsablauf 1x Reset
	Q_bGrdstAblEnde	:BOOL;	//Grundstellungsablauf Ausgeführt

	Q_bDatenLoeschen	:BOOL;	// Ein vorhandener Datensatz soll gelöscht werden
	 
	Q_bGrdstStep1Akt	:BOOL;	// Ist TRUE sobald die Grundstellung aktiv ist. Wenn der Parameter I_bParamEinzelschritte aktiv ist, dann wirds FALSE wenn der nächste Schritt aktiv ist.
	Q_bGrdstStep2Akt	:BOOL;	// Ist TRUE sobald die Weiterschaltbedingung vom vorherigen TRUE ist. Wenn der Parameter I_bParamEinzelschritte aktiv ist, dann wirds FALSE wenn der nächste Schritt aktiv ist.
	Q_bGrdstStep3Akt	:BOOL;	// Ist TRUE sobald die Weiterschaltbedingung vom vorherigen TRUE ist. Wenn der Parameter I_bParamEinzelschritte aktiv ist, dann wirds FALSE wenn der nächste Schritt aktiv ist.
	Q_bGrdstStep4Akt	:BOOL;	// Ist TRUE sobald die Weiterschaltbedingung vom vorherigen TRUE ist. Wenn der Parameter I_bParamEinzelschritte aktiv ist, dann wirds FALSE wenn der nächste Schritt aktiv ist.
	Q_bGrdstStep5Akt	:BOOL;	// Ist TRUE sobald die Weiterschaltbedingung vom vorherigen TRUE ist. Wenn der Parameter I_bParamEinzelschritte aktiv ist, dann wirds FALSE wenn der nächste Schritt aktiv ist.
	Q_bGrdstStep6Akt	:BOOL;	// Ist TRUE sobald die Weiterschaltbedingung vom vorherigen TRUE ist. Wenn der Parameter I_bParamEinzelschritte aktiv ist, dann wirds FALSE wenn der nächste Schritt aktiv ist.
	Q_bGrdstStep7Akt	:BOOL;	// Ist TRUE sobald die Weiterschaltbedingung vom vorherigen TRUE ist. Wenn der Parameter I_bParamEinzelschritte aktiv ist, dann wirds FALSE wenn der nächste Schritt aktiv ist.
	Q_bGrdstStep8Akt	:BOOL;	// Ist TRUE sobald die Weiterschaltbedingung vom vorherigen TRUE ist. Wenn der Parameter I_bParamEinzelschritte aktiv ist, dann wirds FALSE wenn der nächste Schritt aktiv ist.
	Q_bGrdstStep9Akt	:BOOL;	// Ist TRUE sobald die Weiterschaltbedingung vom vorherigen TRUE ist. Dieser Schritt bleibt solange TRUE wie die Grundstellung aktiv ist.

	Q_bGrdstlgMeldg	:BOOL;	// Grundstellung-Meldung für Paneltaste, Softkey etc. mit Blinktakt wenn aktiv. Durchgehen TRUE, wenn Grundstellung Ende
END_VAR
VAR

	rtrigImpAnAbw		:R_TRIG;
	rtrigDatenLoeschen:R_TRIG;
	rTrigAnwahl			:R_TRIG;
	
	bGrdst1xAngw		:BOOL;	// Anwahl der Grundstellung über die Grundstellung-Stations-Anwahl speichern.
	
	nStepState			:INT;
END_VAR

	(*Uni.- Grundstellungsablauf*)
	
	(**************************************************)	
	(*Grundstellung An.-Abwahl*)

	a_AnAbwahl();
	
	(**************************************************)	
	(*Grundstellung Step-Ablauf*)

	b_StepAblauf();

	(**************************************************)	
	(*Zustände anzeigen*)

	y_ZustAnzg();

	(**************************************************)	
	(*Meldungen ausgeben*)

	z_HinwMeld();
	
	(**************************************************)

ACTION a_AnAbwahl:
	
//****************************************************************************************************
// Grundstellung An.-Abwahl
	
	rtrigDatenLoeschen(CLK:= I_bLoeschDatenPos);
									  
	rtrigImpAnAbw (CLK:= (IQ_stUniAnstgEinzelHMI.stHandFktHMI[1].bySwitch > 0
		 						OR IQ_stUniAnstgGesamtHMI.stHandFktHMI[1].bySwitch > 0
								OR I_bGrdstlgAnwTast
								OR (I_bGrdstlgAnfStat
									 AND NOT bGrdst1xAngw) 
								OR (NOT I_bGrdstlgAnfStat
									 AND bGrdst1xAngw))
								AND (I_bGrdstAnwahlFrg
									 AND I_bHandbetrAktiv));

//****************************************************************************************************
//ToDo teilweise nur Anwahl /direkter zugriff auf Teileverfolgung...

	Q_bGrdstAblReset:= FALSE;
	
	IF NOT I_bHandbetrAktiv
		THEN
			Q_bGrdstAblAktiv:= FALSE;
			bGrdst1xAngw	 := FALSE;	
			nStepState		 := 0;			
	ELSIF rtrigImpAnAbw.Q
		THEN
			Q_bGrdstAblAktiv:= NOT Q_bGrdstAblAktiv;
			Q_bGrdstAblReset:= Q_bGrdstAblAktiv;
			bGrdst1xAngw	 := I_bGrdstlgAnfStat;	// Anwahl der Grundstellung über die Grundstellung-Stations-Anwahl speichern
			nStepState		 := 0;
			
	ELSIF rtrigDatenLoeschen.Q
		OR (I_bLoeschDatenPos
			AND NOT Q_bGrdstAblAktiv)
		THEN
			Q_bGrdstAblAktiv	:= TRUE;
			Q_bGrdstAblReset:= Q_bGrdstAblAktiv;
			nStepState		 := 0;
	END_IF

	rTrigAnwahl(CLK := IQ_stUniAnstgBereichHMI.stHandFktHMI[1].bySwitch > 0);
	
	IF rTrigAnwahl.Q
	THEN	// Mit der Bereich-Schnittstelle wird die Grundstellung "nur" gestartet, Nie Gestoppt
		Q_bGrdstAblAktiv	:= TRUE;
		Q_bGrdstAblReset	:= TRUE;
		nStepState		 	:= 0;
	END_IF

//****************************************************************************************************
END_ACTION

ACTION b_StepAblauf:
	
//****************************************************************************************************
// Grundstellung Step-Ablauf

	CASE nStepState OF
0:	//Initialisierung

	Q_bDatenLoeschen:=	
	Q_bGrdstStep1Akt:=
	Q_bGrdstStep2Akt:=
	Q_bGrdstStep3Akt:=
	Q_bGrdstStep4Akt:=
	Q_bGrdstStep5Akt:=
	Q_bGrdstStep6Akt:=
	Q_bGrdstStep7Akt:=
	Q_bGrdstStep8Akt:=
	Q_bGrdstStep9Akt:= FALSE;

	IF Q_bGrdstAblAktiv THEN
		nStepState:= 1;
	END_IF
	
1:	//Ablauf Step 1
	Q_bGrdstStep1Akt:= TRUE;
	
	IF I_bGrdstStep1End THEN
		nStepState:= 2;
		Q_bGrdstStep1Akt	:= NOT I_bParamEinzelschritte;
	END_IF
	
2:	//Ablauf Step 2
	Q_bGrdstStep2Akt:= TRUE;
	
	IF I_bGrdstStep2End THEN
		nStepState:= 3;
		Q_bGrdstStep2Akt	:= NOT I_bParamEinzelschritte;
	END_IF
	
3:	//Ablauf Step 3
	Q_bGrdstStep3Akt:= TRUE;
	
	IF I_bGrdstStep3End THEN
		nStepState:= 4;
		Q_bGrdstStep3Akt	:= NOT I_bParamEinzelschritte;
	END_IF
	
4:	//Ablauf Step 4
	Q_bGrdstStep4Akt:= TRUE;
	
	IF I_bGrdstStep4End THEN
		nStepState:= 5;
		Q_bGrdstStep4Akt	:= NOT I_bParamEinzelschritte;
	END_IF
	
5:	//Ablauf Step 5
	Q_bGrdstStep5Akt:= TRUE;
	
	IF I_bGrdstStep5End THEN
		nStepState:= 6;
		Q_bGrdstStep5Akt	:= NOT I_bParamEinzelschritte;
	END_IF
	
6:	//Ablauf Step 6
	Q_bGrdstStep6Akt:= TRUE;
	
	IF I_bGrdstStep6End THEN
		nStepState:= 7;
		Q_bGrdstStep6Akt	:= NOT I_bParamEinzelschritte;
	END_IF
	
7:	//Ablauf Step 7
	Q_bGrdstStep7Akt:= TRUE;
	
	IF I_bGrdstStep7End THEN
		nStepState:= 8;
		Q_bGrdstStep7Akt	:= NOT I_bParamEinzelschritte;
	END_IF
	
8:	//Ablauf Step 8
	Q_bGrdstStep8Akt:= TRUE;
	
	IF I_bGrdstStep8End THEN
		nStepState:= 9;
		Q_bGrdstStep8Akt	:= NOT I_bParamEinzelschritte;
	END_IF
	
9:	//Ablauf Step 9
	Q_bGrdstStep9Akt:= TRUE;
	
	IF I_bGrdstStep9End THEN
		nStepState:= 10;
	END_IF
	
10://Datenabfrage, wenn Daten zum löschen vorhanden sind, bleibt das Lösch-Bit an
	
	IF I_bDatenVorh
		THEN
			Q_bDatenLoeschen	:= TRUE;	
		ELSE
			Q_bDatenLoeschen	:= FALSE;
			nStepState:= 99;
   END_IF

99://Ablaufende	

	END_CASE	

//****************************************************************************************************

	Q_bGrdstAblEnde:= nStepState = 99
							AND I_bSensPosFreiErk; 
//****************************************************************************************************
END_ACTION

ACTION y_ZustAnzg:
	
//****************************************************************************************************
// Zustände anzeigen

	IF I_bGrdstAnwahlFrg
		AND I_bHandbetrAktiv
	THEN	// Funktion freigegeben
		IQ_stUniAnstgEinzelHMI.stHandFktHMI[1].sColour	:= cDefaultAsString;
		IQ_stUniAnstgEinzelHMI.stHandFktHMI[1].sText		:= 'ausführen';
		IQ_stUniAnstgGesamtHMI.stHandFktHMI[1].sColour	:= cDefaultAsString;
		IQ_stUniAnstgGesamtHMI.stHandFktHMI[1].sText		:= 'ausführen';
		IQ_stUniAnstgBereichHMI.stHandFktHMI[1].sColour	:= cDefaultAsString;
		IQ_stUniAnstgBereichHMI.stHandFktHMI[1].sText	:= 'ausführen';
		IQ_stUniAnstgEinzelHMI.stHandFktHMI[1].byStatus		:= 0;
		IQ_stUniAnstgGesamtHMI.stHandFktHMI[1].byStatus		:= 0;
		IQ_stUniAnstgBereichHMI.stHandFktHMI[1].byStatus	:= 0;
		IQ_stUniAnstgEinzelHMI.stHandFktHMI[1].iDisplayMode	:= 0;
		IQ_stUniAnstgGesamtHMI.stHandFktHMI[1].iDisplayMode	:= 0;
		IQ_stUniAnstgBereichHMI.stHandFktHMI[1].iDisplayMode	:= 0;

		IF Q_bGrdstAblAktiv
			AND NOT Q_bGrdstAblEnde
		THEN	// Handfunktion aktiv			
			IQ_stUniAnstgEinzelHMI.stHandFktHMI[1].sColour	:= cGelbAsString;
			IQ_stUniAnstgEinzelHMI.stHandFktHMI[1].sText		:= 'ausführen';
			IQ_stUniAnstgGesamtHMI.stHandFktHMI[1].sColour	:= cGelbAsString;
			IQ_stUniAnstgGesamtHMI.stHandFktHMI[1].sText		:= 'ausführen';
			IQ_stUniAnstgBereichHMI.stHandFktHMI[1].sColour	:= cGelbAsString;
			IQ_stUniAnstgBereichHMI.stHandFktHMI[1].sText	:= 'ausführen';
			IQ_stUniAnstgEinzelHMI.stHandFktHMI[1].byStatus		:= 0;
			IQ_stUniAnstgGesamtHMI.stHandFktHMI[1].byStatus		:= 0;
			IQ_stUniAnstgBereichHMI.stHandFktHMI[1].byStatus	:= 0;
			IQ_stUniAnstgEinzelHMI.stHandFktHMI[1].iDisplayMode	:= 2;
			IQ_stUniAnstgGesamtHMI.stHandFktHMI[1].iDisplayMode	:= 2;
			IQ_stUniAnstgBereichHMI.stHandFktHMI[1].iDisplayMode	:= 2;
		END_IF
		
		IF Q_bGrdstAblEnde
		THEN	// Handfunktion ausgeführt
			IQ_stUniAnstgEinzelHMI.stHandFktHMI[1].sColour	:= cGruenAsString;
			IQ_stUniAnstgEinzelHMI.stHandFktHMI[1].sText		:= 'ausgeführt';
			IQ_stUniAnstgGesamtHMI.stHandFktHMI[1].sColour	:= cGruenAsString;
			IQ_stUniAnstgGesamtHMI.stHandFktHMI[1].sText		:= 'ausgeführt';
			IQ_stUniAnstgBereichHMI.stHandFktHMI[1].sColour	:= cGruenAsString;
			IQ_stUniAnstgBereichHMI.stHandFktHMI[1].sText	:= 'ausgeführt';
			IQ_stUniAnstgEinzelHMI.stHandFktHMI[1].byStatus		:= 0;
			IQ_stUniAnstgGesamtHMI.stHandFktHMI[1].byStatus		:= 0;
			IQ_stUniAnstgBereichHMI.stHandFktHMI[1].byStatus	:= 0;
			IQ_stUniAnstgEinzelHMI.stHandFktHMI[1].iDisplayMode	:= 0;
			IQ_stUniAnstgGesamtHMI.stHandFktHMI[1].iDisplayMode	:= 0;
			IQ_stUniAnstgBereichHMI.stHandFktHMI[1].iDisplayMode	:= 0;
		END_IF
		
	ELSE	// Funktion gesperrt
		IQ_stUniAnstgEinzelHMI.stHandFktHMI[1].sColour	:= cDefaultAsString;
		IQ_stUniAnstgEinzelHMI.stHandFktHMI[1].sText		:= 'ausführen';
		IQ_stUniAnstgGesamtHMI.stHandFktHMI[1].sColour	:= cDefaultAsString;
		IQ_stUniAnstgGesamtHMI.stHandFktHMI[1].sText		:= 'ausführen';
		IQ_stUniAnstgBereichHMI.stHandFktHMI[1].sColour	:= cDefaultAsString;
		IQ_stUniAnstgBereichHMI.stHandFktHMI[1].sText	:= 'ausführen';
		IQ_stUniAnstgEinzelHMI.stHandFktHMI[1].byStatus		:= 1;
		IQ_stUniAnstgGesamtHMI.stHandFktHMI[1].byStatus		:= 1;
		IQ_stUniAnstgBereichHMI.stHandFktHMI[1].byStatus	:= 1;
		IQ_stUniAnstgEinzelHMI.stHandFktHMI[1].iDisplayMode	:= 0;
		IQ_stUniAnstgGesamtHMI.stHandFktHMI[1].iDisplayMode	:= 0;
		IQ_stUniAnstgBereichHMI.stHandFktHMI[1].iDisplayMode	:= 0;
	END_IF
	
// Der Zustand in der Bereichsschnittstelle wird ggf. nicht korrekt angezeigt.
//	IQ_stUniAnstgBereichHMI.stHandFktHMI[1].byStatus:= 0;
END_ACTION

ACTION z_HinwMeld:

//****************************************************************************************************
// Fehler-Meldungen ausgeben
	
	// Die beiden Ein-Ausgangsvariablen IQ_stUniAnstgBereichHMI und IQ_stUniAnstgGesamtHMI werden hier nicht bespielt, weil sich die Meldungen sonst doppeln würden.

	IQ_stUniAnstgEinzelHMI.stMeldAusgHMI.SourceID		:= 0;	// Nicht mehr verwendet
	IQ_stUniAnstgEinzelHMI.stMeldAusgHMI.SourceName		:= I_sStatName;

	IF bTestMeldGrdstlg
	THEN	// Testmeldung für alle Grundstellungsmeldungen
		IQ_stUniAnstgEinzelHMI.stMeldAusgHMI.bMeldAktiv					:=
		IQ_stUniAnstgEinzelHMI.stMeldAusgHMI.bMeldDonemitEntnahme	:= 
		IQ_stUniAnstgEinzelHMI.stMeldAusgHMI.bMeldDoneOhneEntnahme	:= TRUE;
	ELSIF nStepState >= 1
	THEN
		IQ_stUniAnstgEinzelHMI.stMeldAusgHMI.bMeldAktiv					:= TRUE; 
		IQ_stUniAnstgEinzelHMI.stMeldAusgHMI.bMeldDonemitEntnahme	:= FALSE;
		IQ_stUniAnstgEinzelHMI.stMeldAusgHMI.bMeldDoneOhneEntnahme	:= FALSE;
		IF nStepState >= 10
		THEN
			IQ_stUniAnstgEinzelHMI.stMeldAusgHMI.bMeldAktiv			:= FALSE;
			IF I_bTeileEntnahmeNoetig
			THEN 
				IQ_stUniAnstgEinzelHMI.stMeldAusgHMI.bMeldDonemitEntnahme	:= TRUE;
			ELSE 
				IQ_stUniAnstgEinzelHMI.stMeldAusgHMI.bMeldDoneOhneEntnahme	:= TRUE;
			END_IF
		END_IF
	ELSE
		IQ_stUniAnstgEinzelHMI.stMeldAusgHMI.bMeldAktiv						:=
		IQ_stUniAnstgEinzelHMI.stMeldAusgHMI.bMeldDonemitEntnahme		:= 
		IQ_stUniAnstgEinzelHMI.stMeldAusgHMI.bMeldDoneOhneEntnahme		:= FALSE;
   END_IF

//****************************************************************************************************
// Hardware-Meldungen

	Q_bGrdstlgMeldg:= (Q_bGrdstAblAktiv AND bTaktLangsam) OR	Q_bGrdstAblEnde;

//****************************************************************************************************
END_ACTION

END_FUNCTION_BLOCK

// POUs/Grundstellung/FB_UniGrdstlgAblGesamt
// Dieser Grundstellungsablauf hat noch einen zusätzlichen Ein-Ausgang für einen Grundstellungsbereich (z.B. einen Schutzbereich)
// und für die HMI-Taste Grundstellung Gesamt.
// Das Ganze verhält sich aber so, dass die VAR_IN_OUT für Bereich und Gesamt dann von allen Grundstellungsabläufen beschrieben wird, an die diese Strukturen angelegt werden.
// Somit wird nur der Zustand vom letzten Grundstellungsablauf, an dem diese Strukturen angelegt sind, angezeigt.
// hat aber sonst die gleiche Funktion wie der FB_UniGrdstlgAbl
FUNCTION_BLOCK FB_UniGrdstlgAblGesamt
VAR_INPUT

	I_sStatName			:Tc2_System.T_MaxString;	// Aktueller Stationsname für Fehlermeldungen

	I_bHandbetrAktiv	:BOOL;	// Betriebsart, Schutzbereich etc.
	I_bGrdstAnwahlFrg	:BOOL;	// Betriebsart, Schutzbereich etc.

	I_bLoeschDatenPos :BOOL;	// Grundstellungsablauf-Anwahl durch Datensatz löschen in der Teileverfolgung
	I_bGrdstlgAnwTast :BOOL;	// Grundstellungsablauf-Anwahl durch Paneltaste, Softkey etc.
	I_bGrdstlgAnfStat	:BOOL;	// Grundstellungsablauf-Anwahl durch extern z.B. Referenzablauf. Bei fallender Flanke wird die Grundstellung wieder abgewählt, bzw. umgeschaltet
	
	I_bDatenVorh		:BOOL;	// Sind Daten vorhanden wird das Lösch-Bit gesetzt
	I_bSensPosFreiErk	:BOOL:= TRUE;	// Optional: Erkennung Teileentnahme. Grundstellung ist erst zuende, wenn dieses Bit TRUE ist.
	I_bTeileEntnahmeNoetig	: BOOL;	// Nur für eine Melden, dass nach der erfolgreichen Grundstellungsfahrt das Teil entnommen werden soll. Die Meldung bleibt so lange an wie die Grundstellung aktiv ist oder dieses Bit gesetzt
	 
	I_bGrdstStep1End	:BOOL:= TRUE;	// Rückmeldung Schritt 1 fertig
	I_bGrdstStep2End	:BOOL:= TRUE;	// Rückmeldung Schritt 2 fertig
	I_bGrdstStep3End	:BOOL:= TRUE;	// Rückmeldung Schritt 3 fertig
	I_bGrdstStep4End	:BOOL:= TRUE;	// Rückmeldung Schritt 4 fertig
	I_bGrdstStep5End	:BOOL:= TRUE;	// Rückmeldung Schritt 5 fertig
	I_bGrdstStep6End	:BOOL:= TRUE;	// Rückmeldung Schritt 6 fertig
	I_bGrdstStep7End	:BOOL:= TRUE;	// Rückmeldung Schritt 7 fertig
	I_bGrdstStep8End	:BOOL:= TRUE;	// Rückmeldung Schritt 8 fertig
	I_bGrdstStep9End	:BOOL:= TRUE;	// Rückmeldung Schritt 9 fertig

	I_bParamEinzelschritte	: BOOL;	// Wenn dieser Parameter an ist, dann sind die Schritte nur einzeln an. Also wenn Q_bGrdstStep2Akt an geht, geht Q_bGrdstStep1Akt aus.

END_VAR
VAR_IN_OUT
	IQ_stUniAnstgStation	:ST_UniGrdstlgAbl;	//HMI-Struktur Einzelposition
	IQ_stUniAnstgBereich	:ST_UniGrdstlgAbl;	//HMI-Struktur für einen Bereich, z.B. Schutzbereich. Über diese Schnittstelle ist nur einschalten möglich, nicht ausschalten. Es wird nur der Zustand von dem letzten Grundstellungsablauf mit dieser Schnittstelle angezeigt.
	IQ_stUniAnstgGesamt	:ST_UniGrdstlgAbl;	//HMI-Struktur Grundstellung Gesamt.  Über diese Schnittstelle ist nur einschalten möglich, nicht ausschalten. Es wird nur der Zustand von dem letzten Grundstellungsablauf mit dieser Schnittstelle angezeigt.
	IQ_stUniAnstgListe	:ST_UniGrdstlgAbl;	//HMI-Struktur Anlagenbereich/Gesamtanlage, Liste mit allen Grundstellungsabläufen
END_VAR
VAR_OUTPUT
	Q_bGrdstAblAktiv	:BOOL;	// Gesamtablauf Aktiv
	Q_bGrdstAblReset	:BOOL;	// Gesamtablauf 1x Reset
	Q_bGrdstAblEnde	:BOOL;	// Gesamtablauf Ausgeführt
	
	Q_bDatenLoeschen	:BOOL;	// Ein vorhandener Datensatz soll gelöscht werden
	 
	Q_bGrdstStep1Akt	:BOOL;	// Ist TRUE sobald die Grundstellung aktiv ist. Wenn der Parameter I_bParamEinzelschritte aktiv ist, dann wirds FALSE wenn der nächste Schritt aktiv ist.
	Q_bGrdstStep2Akt	:BOOL;	// Ist TRUE sobald die Weiterschaltbedingung vom vorherigen TRUE ist. Wenn der Parameter I_bParamEinzelschritte aktiv ist, dann wirds FALSE wenn der nächste Schritt aktiv ist.
	Q_bGrdstStep3Akt	:BOOL;	// Ist TRUE sobald die Weiterschaltbedingung vom vorherigen TRUE ist. Wenn der Parameter I_bParamEinzelschritte aktiv ist, dann wirds FALSE wenn der nächste Schritt aktiv ist.
	Q_bGrdstStep4Akt	:BOOL;	// Ist TRUE sobald die Weiterschaltbedingung vom vorherigen TRUE ist. Wenn der Parameter I_bParamEinzelschritte aktiv ist, dann wirds FALSE wenn der nächste Schritt aktiv ist.
	Q_bGrdstStep5Akt	:BOOL;	// Ist TRUE sobald die Weiterschaltbedingung vom vorherigen TRUE ist. Wenn der Parameter I_bParamEinzelschritte aktiv ist, dann wirds FALSE wenn der nächste Schritt aktiv ist.
	Q_bGrdstStep6Akt	:BOOL;	// Ist TRUE sobald die Weiterschaltbedingung vom vorherigen TRUE ist. Wenn der Parameter I_bParamEinzelschritte aktiv ist, dann wirds FALSE wenn der nächste Schritt aktiv ist.
	Q_bGrdstStep7Akt	:BOOL;	// Ist TRUE sobald die Weiterschaltbedingung vom vorherigen TRUE ist. Wenn der Parameter I_bParamEinzelschritte aktiv ist, dann wirds FALSE wenn der nächste Schritt aktiv ist.
	Q_bGrdstStep8Akt	:BOOL;	// Ist TRUE sobald die Weiterschaltbedingung vom vorherigen TRUE ist. Wenn der Parameter I_bParamEinzelschritte aktiv ist, dann wirds FALSE wenn der nächste Schritt aktiv ist.
	Q_bGrdstStep9Akt	:BOOL;	// Ist TRUE sobald die Weiterschaltbedingung vom vorherigen TRUE ist. Dieser Schritt bleibt solange TRUE wie die Grundstellung aktiv ist.

	Q_bGrdstlgMeldg	:BOOL;	// Grundstellung-Meldung für Paneltaste, Softkey etc. mit Blinktakt wenn aktiv. Durchgehen TRUE, wenn Grundstellung Ende
END_VAR
VAR

	rtrigImpAnAbw		:R_TRIG;
	rtrigDatenLoeschen:R_TRIG;
	rTrigAnwahl			:R_TRIG;
	
	bGrdst1xAngw		:BOOL;	// Anwahl der Grundstellung über die Grundstellung-Stations-Anwahl speichern.
	
	nStepState			:INT;
END_VAR

	(*Uni.- Grundstellungsablauf*)
	
	(**************************************************)	
	(*Grundstellung An.-Abwahl*)

	a_AnAbwahl();
	
	(**************************************************)	
	(*Grundstellung Step-Ablauf*)

	b_StepAblauf();

	(**************************************************)	
	(*Zustände anzeigen*)

	y_ZustAnzg();

	(**************************************************)	
	(*Meldungen ausgeben*)

	z_HinwMeld();
	
	(**************************************************)

ACTION a_AnAbwahl:
	
//****************************************************************************************************
// Grundstellung An.-Abwahl
	
	rtrigDatenLoeschen(CLK:= I_bLoeschDatenPos);
									  
	rtrigImpAnAbw (CLK:= (IQ_stUniAnstgStation.stHandFktHMI[1].bySwitch > 0
		 						OR IQ_stUniAnstgListe.stHandFktHMI[1].bySwitch > 0
								OR I_bGrdstlgAnwTast
								OR (I_bGrdstlgAnfStat
									 AND NOT bGrdst1xAngw) 
								OR (NOT I_bGrdstlgAnfStat
									 AND bGrdst1xAngw))
								AND (I_bGrdstAnwahlFrg
									 AND I_bHandbetrAktiv));

//****************************************************************************************************
//ToDo teilweise nur Anwahl /direkter zugriff auf Teileverfolgung...

	Q_bGrdstAblReset:= FALSE;
	
	IF NOT I_bHandbetrAktiv
		THEN
			Q_bGrdstAblAktiv:= FALSE;
			bGrdst1xAngw	 := FALSE;	
			nStepState		 := 0;			
	ELSIF rtrigImpAnAbw.Q
		THEN
			Q_bGrdstAblAktiv:= NOT Q_bGrdstAblAktiv;
			Q_bGrdstAblReset:= Q_bGrdstAblAktiv;
			bGrdst1xAngw	 := I_bGrdstlgAnfStat;	// Anwahl der Grundstellung über die Grundstellung-Stations-Anwahl speichern
			nStepState		 := 0;
			
	ELSIF rtrigDatenLoeschen.Q
		OR (I_bLoeschDatenPos
			AND NOT Q_bGrdstAblAktiv)
		THEN
			Q_bGrdstAblAktiv	:= TRUE;
			Q_bGrdstAblReset:= Q_bGrdstAblAktiv;
			nStepState		 := 0;
	END_IF

	rTrigAnwahl(CLK :=
		IQ_stUniAnstgBereich.stHandFktHMI[1].bySwitch > 0
		OR IQ_stUniAnstgGesamt.stHandFktHMI[1].bySwitch > 0);
	
	IF rTrigAnwahl.Q
	THEN	// Mit diesen Schnittstellen wird die Grundstellung "nur" gestartet, Nie Gestoppt
		Q_bGrdstAblAktiv	:= TRUE;
		Q_bGrdstAblReset	:= TRUE;
		nStepState		 	:= 0;
	END_IF

//****************************************************************************************************
END_ACTION

ACTION b_StepAblauf:
	
//****************************************************************************************************
// Grundstellung Step-Ablauf

	CASE nStepState OF
0:	//Initialisierung

	Q_bDatenLoeschen:=	
	Q_bGrdstStep1Akt:=
	Q_bGrdstStep2Akt:=
	Q_bGrdstStep3Akt:=
	Q_bGrdstStep4Akt:=
	Q_bGrdstStep5Akt:=
	Q_bGrdstStep6Akt:=
	Q_bGrdstStep7Akt:=
	Q_bGrdstStep8Akt:=
	Q_bGrdstStep9Akt:= FALSE;

	IF Q_bGrdstAblAktiv THEN
		nStepState:= 1;
	END_IF
	
1:	//Ablauf Step 1
	Q_bGrdstStep1Akt:= TRUE;
	
	IF I_bGrdstStep1End THEN
		nStepState:= 2;
		Q_bGrdstStep1Akt	:= NOT I_bParamEinzelschritte;
	END_IF
	
2:	//Ablauf Step 2
	Q_bGrdstStep2Akt:= TRUE;
	
	IF I_bGrdstStep2End THEN
		nStepState:= 3;
		Q_bGrdstStep2Akt	:= NOT I_bParamEinzelschritte;
	END_IF
	
3:	//Ablauf Step 3
	Q_bGrdstStep3Akt:= TRUE;
	
	IF I_bGrdstStep3End THEN
		nStepState:= 4;
		Q_bGrdstStep3Akt	:= NOT I_bParamEinzelschritte;
	END_IF
	
4:	//Ablauf Step 4
	Q_bGrdstStep4Akt:= TRUE;
	
	IF I_bGrdstStep4End THEN
		nStepState:= 5;
		Q_bGrdstStep4Akt	:= NOT I_bParamEinzelschritte;
	END_IF
	
5:	//Ablauf Step 5
	Q_bGrdstStep5Akt:= TRUE;
	
	IF I_bGrdstStep5End THEN
		nStepState:= 6;
		Q_bGrdstStep5Akt	:= NOT I_bParamEinzelschritte;
	END_IF
	
6:	//Ablauf Step 6
	Q_bGrdstStep6Akt:= TRUE;
	
	IF I_bGrdstStep6End THEN
		nStepState:= 7;
		Q_bGrdstStep6Akt	:= NOT I_bParamEinzelschritte;
	END_IF
	
7:	//Ablauf Step 7
	Q_bGrdstStep7Akt:= TRUE;
	
	IF I_bGrdstStep7End THEN
		nStepState:= 8;
		Q_bGrdstStep7Akt	:= NOT I_bParamEinzelschritte;
	END_IF
	
8:	//Ablauf Step 8
	Q_bGrdstStep8Akt:= TRUE;
	
	IF I_bGrdstStep8End THEN
		nStepState:= 9;
		Q_bGrdstStep8Akt	:= NOT I_bParamEinzelschritte;
	END_IF
	
9:	//Ablauf Step 9
	Q_bGrdstStep9Akt:= TRUE;
	
	IF I_bGrdstStep9End THEN
		nStepState:= 10;
	END_IF
	
10://Datenabfrage, wenn Daten zum löschen vorhanden sind, bleibt das Lösch-Bit an
	
	IF I_bDatenVorh
		THEN
			Q_bDatenLoeschen	:= TRUE;	
		ELSE
			Q_bDatenLoeschen	:= FALSE;
			nStepState:= 99;
   END_IF

99://Ablaufende	

	END_CASE	

//****************************************************************************************************

	Q_bGrdstAblEnde:= nStepState = 99
							AND I_bSensPosFreiErk;

//****************************************************************************************************
END_ACTION

ACTION y_ZustAnzg:
	
//****************************************************************************************************
// Zustände anzeigen

	IF I_bGrdstAnwahlFrg
		AND I_bHandbetrAktiv
	THEN	// Funktion freigegeben
		IQ_stUniAnstgStation.stHandFktHMI[1].sColour	:= cDefaultAsString;
		IQ_stUniAnstgStation.stHandFktHMI[1].sText	:= 'ausführen';
		IQ_stUniAnstgListe.stHandFktHMI[1].sColour	:= cDefaultAsString;
		IQ_stUniAnstgListe.stHandFktHMI[1].sText		:= 'ausführen';
		IQ_stUniAnstgBereich.stHandFktHMI[1].sColour	:= cDefaultAsString;
		IQ_stUniAnstgBereich.stHandFktHMI[1].sText	:= 'ausführen';
		IQ_stUniAnstgGesamt.stHandFktHMI[1].sColour	:= cDefaultAsString;
		IQ_stUniAnstgGesamt.stHandFktHMI[1].sText		:= 'ausführen';
		IQ_stUniAnstgStation.stHandFktHMI[1].byStatus	:= 0;
		IQ_stUniAnstgListe.stHandFktHMI[1].byStatus		:= 0;
		IQ_stUniAnstgBereich.stHandFktHMI[1].byStatus	:= 0;
		IQ_stUniAnstgGesamt.stHandFktHMI[1].byStatus		:= 0;
		IQ_stUniAnstgListe.stHandFktHMI[1].iDisplayMode		:= 0;
		IQ_stUniAnstgStation.stHandFktHMI[1].iDisplayMode	:= 0;
		IQ_stUniAnstgBereich.stHandFktHMI[1].iDisplayMode	:= 0;
		IQ_stUniAnstgGesamt.stHandFktHMI[1].iDisplayMode	:= 0;

		IF Q_bGrdstAblAktiv
			AND NOT Q_bGrdstAblEnde
		THEN	// Handfunktion aktiv			
			IQ_stUniAnstgStation.stHandFktHMI[1].sColour	:= cGelbAsString;
			IQ_stUniAnstgStation.stHandFktHMI[1].sText	:= 'ausführen';
			IQ_stUniAnstgListe.stHandFktHMI[1].sColour	:= cGelbAsString;
			IQ_stUniAnstgListe.stHandFktHMI[1].sText		:= 'ausführen';
			IQ_stUniAnstgBereich.stHandFktHMI[1].sColour	:= cGelbAsString;
			IQ_stUniAnstgBereich.stHandFktHMI[1].sText	:= 'ausführen';
			IQ_stUniAnstgGesamt.stHandFktHMI[1].sColour	:= cGelbAsString;
			IQ_stUniAnstgGesamt.stHandFktHMI[1].sText		:= 'ausführen';
			IQ_stUniAnstgStation.stHandFktHMI[1].byStatus	:= 0;
			IQ_stUniAnstgListe.stHandFktHMI[1].byStatus		:= 0;
			IQ_stUniAnstgBereich.stHandFktHMI[1].byStatus	:= 0;
			IQ_stUniAnstgGesamt.stHandFktHMI[1].byStatus		:= 0;
			IQ_stUniAnstgListe.stHandFktHMI[1].iDisplayMode		:= 2;
			IQ_stUniAnstgStation.stHandFktHMI[1].iDisplayMode	:= 2;
			IQ_stUniAnstgBereich.stHandFktHMI[1].iDisplayMode	:= 2;
			IQ_stUniAnstgGesamt.stHandFktHMI[1].iDisplayMode	:= 2;
		END_IF
		
		IF Q_bGrdstAblEnde
		THEN	// Handfunktion ausgeführt
			IQ_stUniAnstgStation.stHandFktHMI[1].sColour	:= cGruenAsString;
			IQ_stUniAnstgStation.stHandFktHMI[1].sText	:= 'ausgeführt';
			IQ_stUniAnstgListe.stHandFktHMI[1].sColour	:= cGruenAsString;
			IQ_stUniAnstgListe.stHandFktHMI[1].sText		:= 'ausgeführt';
			IQ_stUniAnstgBereich.stHandFktHMI[1].sColour	:= cGruenAsString;
			IQ_stUniAnstgBereich.stHandFktHMI[1].sText	:= 'ausgeführt';
			IQ_stUniAnstgGesamt.stHandFktHMI[1].sColour	:= cGruenAsString;
			IQ_stUniAnstgGesamt.stHandFktHMI[1].sText		:= 'ausgeführt';
			IQ_stUniAnstgStation.stHandFktHMI[1].byStatus	:= 0;
			IQ_stUniAnstgListe.stHandFktHMI[1].byStatus		:= 0;
			IQ_stUniAnstgBereich.stHandFktHMI[1].byStatus	:= 0;
			IQ_stUniAnstgGesamt.stHandFktHMI[1].byStatus		:= 0;
			IQ_stUniAnstgListe.stHandFktHMI[1].iDisplayMode		:= 0;
			IQ_stUniAnstgStation.stHandFktHMI[1].iDisplayMode	:= 0;
			IQ_stUniAnstgBereich.stHandFktHMI[1].iDisplayMode	:= 0;
			IQ_stUniAnstgGesamt.stHandFktHMI[1].iDisplayMode	:= 0;
		END_IF
		
	ELSE	// Funktion gesperrt
		IQ_stUniAnstgStation.stHandFktHMI[1].sColour	:= cDefaultAsString;
		IQ_stUniAnstgStation.stHandFktHMI[1].sText	:= 'ausführen';
		IQ_stUniAnstgListe.stHandFktHMI[1].sColour	:= cDefaultAsString;
		IQ_stUniAnstgListe.stHandFktHMI[1].sText		:= 'ausführen';
		IQ_stUniAnstgBereich.stHandFktHMI[1].sColour	:= cDefaultAsString;
		IQ_stUniAnstgBereich.stHandFktHMI[1].sText	:= 'ausführen';
		IQ_stUniAnstgGesamt.stHandFktHMI[1].sColour	:= cDefaultAsString;
		IQ_stUniAnstgGesamt.stHandFktHMI[1].sText		:= 'ausführen';
		IQ_stUniAnstgStation.stHandFktHMI[1].byStatus	:= 1;
		IQ_stUniAnstgListe.stHandFktHMI[1].byStatus		:= 1;
		IQ_stUniAnstgBereich.stHandFktHMI[1].byStatus	:= 1;
		IQ_stUniAnstgGesamt.stHandFktHMI[1].byStatus		:= 1;
		IQ_stUniAnstgListe.stHandFktHMI[1].iDisplayMode		:= 0;
		IQ_stUniAnstgStation.stHandFktHMI[1].iDisplayMode	:= 0;
		IQ_stUniAnstgBereich.stHandFktHMI[1].iDisplayMode	:= 0;
		IQ_stUniAnstgGesamt.stHandFktHMI[1].iDisplayMode	:= 0;
	END_IF
	
// Der Zustand in der Bereichsschnittstelle wird ggf. nicht korrekt angezeigt.
//	IQ_stUniAnstgBereich.stHandFktHMI[1].byStatus:= 0;
//	IQ_stUniAnstgGesamt.stHandFktHMI[1].byStatus:= 0;
END_ACTION

ACTION z_HinwMeld:

//****************************************************************************************************
// Fehler-Meldungen ausgeben
	
	// Die drei Ein-Ausgangsvariablen IQ_stUniAnstgListe, IQ_stUniAnstgBereich und IQ_stUniAnstgGesamt werden hier nicht bespielt, weil sich die Meldungen sonst doppeln würden.
	
	IQ_stUniAnstgStation.stMeldAusgHMI.SourceID		:= 0;	// Nicht mehr verwendet
	IQ_stUniAnstgStation.stMeldAusgHMI.SourceName	:= I_sStatName;

	IF bTestMeldGrdstlg
	THEN	// Testmeldung für alle Grundstellungsmeldungen
		IQ_stUniAnstgStation.stMeldAusgHMI.bMeldAktiv						:=
		IQ_stUniAnstgStation.stMeldAusgHMI.bMeldDonemitEntnahme		:= 
		IQ_stUniAnstgStation.stMeldAusgHMI.bMeldDoneOhneEntnahme		:= TRUE;
	ELSIF nStepState >= 1
	THEN
		IQ_stUniAnstgStation.stMeldAusgHMI.bMeldAktiv					:= TRUE; 
		IQ_stUniAnstgStation.stMeldAusgHMI.bMeldDonemitEntnahme	:= FALSE;
		IQ_stUniAnstgStation.stMeldAusgHMI.bMeldDoneOhneEntnahme	:= FALSE;
		IF nStepState >= 10
		THEN
			IQ_stUniAnstgStation.stMeldAusgHMI.bMeldAktiv			:= FALSE;
			IF I_bTeileEntnahmeNoetig
			THEN 
				IQ_stUniAnstgStation.stMeldAusgHMI.bMeldDonemitEntnahme	:= TRUE;
			ELSE 
				IQ_stUniAnstgStation.stMeldAusgHMI.bMeldDoneOhneEntnahme	:= TRUE;
			END_IF
		END_IF
	ELSE
		IQ_stUniAnstgStation.stMeldAusgHMI.bMeldAktiv						:=
		IQ_stUniAnstgStation.stMeldAusgHMI.bMeldDonemitEntnahme		:= 
		IQ_stUniAnstgStation.stMeldAusgHMI.bMeldDoneOhneEntnahme		:= FALSE;
   END_IF
		
//****************************************************************************************************
// Hardware-Meldungen

	Q_bGrdstlgMeldg:= (Q_bGrdstAblAktiv AND bTaktLangsam) OR	Q_bGrdstAblEnde;

//****************************************************************************************************
END_ACTION

END_FUNCTION_BLOCK

// POUs/Logging/F_TimeStruct
// Diese Funktion beschreibt den STRING in der Struktur ST_TimeStruct
FUNCTION F_TimeStruct : ST_TimeStruct
VAR_INPUT
	I_stTimeStruct	: Tc2_Utilities.TIMESTRUCT;	// TimeStruct aus Tc2_Utilities.NT_GetTime
	I_sTrennzeichen	: STRING(1)	:= ';';	// Trennzeichen zwischen den Datum und der Uhrzeit für die Verwendung in einer CSV-Datei 
END_VAR
VAR
	sTime	: STRING;
END_VAR

// Die alte Struktur einfach erstmal überschreiben. ST_TimeStamp ist eine Ableitung von Tc2_Utilities.TIMESTRUCT. Daher müsste das klappen
F_TimeStruct.wDay				:= I_stTimeStruct.wDay;
F_TimeStruct.wDayOfWeek		:= I_stTimeStruct.wDayOfWeek;
F_TimeStruct.wHour			:= I_stTimeStruct.wHour;
F_TimeStruct.wMilliseconds	:= I_stTimeStruct.wMilliseconds;
F_TimeStruct.wMinute			:= I_stTimeStruct.wMinute;
F_TimeStruct.wMonth			:= I_stTimeStruct.wMonth;
F_TimeStruct.wSecond			:= I_stTimeStruct.wSecond;
F_TimeStruct.wYear			:= I_stTimeStruct.wYear;

//************************************************************************************************************
// ggf Hochkomma wenn CSV-Datei
sTime := CONCAT(sTime,';');

//************************************************************************************************************
// Tag
IF I_stTimeStruct.wDay < 10
THEN
	sTime := CONCAT(sTime,'0');
END_IF
sTime := CONCAT(sTime,WORD_TO_STRING(I_stTimeStruct.wDay));
sTime := CONCAT(sTime,'-');

//************************************************************************************************************
// Monat
IF I_stTimeStruct.wMonth < 10
THEN
	sTime := CONCAT(sTime,'0');
END_IF
sTime := CONCAT(sTime,WORD_TO_STRING(I_stTimeStruct.wMonth));
sTime := CONCAT(sTime,'-');

//************************************************************************************************************
// Jahr
sTime := CONCAT(sTime,WORD_TO_STRING(I_stTimeStruct.wYear));

//************************************************************************************************************
// Trennung
sTime := CONCAT(sTime,I_sTrennzeichen);

//************************************************************************************************************
// Stunde
IF I_stTimeStruct.wHour < 10
THEN
	sTime := CONCAT(sTime,'0');
END_IF

sTime := CONCAT(sTime,WORD_TO_STRING(I_stTimeStruct.wHour));
sTime := CONCAT(sTime,':');

//************************************************************************************************************
// Minute
IF I_stTimeStruct.wMinute < 10
THEN
	sTime := CONCAT(sTime,'0');
END_IF

sTime := CONCAT(sTime,WORD_TO_STRING(I_stTimeStruct.wMinute));
sTime := CONCAT(sTime,':');

//************************************************************************************************************
// Sekunde
IF I_stTimeStruct.wSecond < 10
THEN
	sTime := CONCAT(sTime,'0');
END_IF

sTime := CONCAT(sTime,WORD_TO_STRING(I_stTimeStruct.wSecond));
sTime := CONCAT(sTime,':');

//************************************************************************************************************
// Millisekunde
IF I_stTimeStruct.wMilliseconds < 10
THEN
	sTime := CONCAT(sTime,'00');
ELSIF I_stTimeStruct.wMilliseconds < 100
THEN
	sTime := CONCAT(sTime,'0');
END_IF

sTime := CONCAT(sTime,WORD_TO_STRING(I_stTimeStruct.wMilliseconds));

//************************************************************************************************************
// Zuweisung
F_TimeStruct.sTimeStamp	:= sTime;

// ENDE

END_FUNCTION

// POUs/Logging/FB_LogToFile
FUNCTION_BLOCK FB_LogToFile
VAR_INPUT
	I_bStart			: BOOL;	

	I_sDateipfad	: T_MaxString;
	I_sDateiname	: T_MaxString;
	I_sUeberschrift: T_MaxString;
	I_sZeile			: T_MaxString;
END_VAR
VAR_OUTPUT
	Q_bDone		: BOOL;
END_VAR
VAR
	nStep			: INT;
	sPfadname	: Tc2_System.T_MaxString;
	sZeile		: Tc2_System.T_MaxString;
	fbFindFile	: Tc2_Utilities.FB_EnumFindFileEntry;
	fbFileOpen 	: Tc2_System.FB_FileOpen;
	fbFileWrite : Tc2_System.FB_FileWrite;
	fbFileClose	: Tc2_System.FB_FileClose;
END_VAR


CASE nStep OF
///////////////////////////////////////////////////////////
0: //INIT
	fbFileOpen(bExecute := FALSE);
	fbFindFile(bExecute := FALSE);
	fbFileWrite(bExecute := FALSE);
	fbFileClose(bExecute := FALSE);
	sPfadname	:= '';
	Q_bDone		:= FALSE;
	IF I_bStart
		AND I_sZeile <> ''
	THEN
		sPfadname :=CONCAT(CONCAT(CONCAT(I_sDateipfad,'\'),I_sDateiname),'.csv');
		nStep := 5;
	END_IF

///////////////////////////////////////////////////////////
5: //Check ob Datei vorhanden ist
	fbFindFile(
		sNetId		:= , 
		sPathName	:= sPfadname, 
		eCmd			:= , 
		bExecute		:= TRUE, 
		tTimeout		:= T#2S, 
		bBusy			=> , 
		bError		=> , 
		nErrID		=> , 
		bEOE			=> , 
		stFindFile	=> );
	
	IF NOT fbFindFile.bBusy
		AND NOT fbFindFile.bError
	THEN
		nStep:= 10;
	END_IF
///////////////////////////////////////////////////////////
10: // Öffne Datei
	fbFileOpen(
		sNetId		:= , 
		sPathName	:= sPfadname, 
		nMode			:= Tc2_System.FOPEN_MODEAPPEND OR Tc2_System.FOPEN_MODEPLUS, 
		ePath			:= Tc2_System.PATH_GENERIC , 
		bExecute		:= TRUE, 
		tTimeout		:= T#2S, 
		bBusy			=> , 
		bError		=> , 
		nErrId		=> , 
		hFile			=> );
		
	IF NOT fbFileOpen.bBusy
		AND NOT fbFileOpen.bError
	THEN
		IF fbFindFile.stFindFile.sFileName <> ''
		THEN
			nStep := 20;
		ELSE
			nStep:= 13;
		END_IF
	END_IF
	
///////////////////////////////////////////////////////////
13: // Schreibe Überschrift
	fbFileWrite(
		sNetId		:= , 
		hFile			:= fbFileOpen.hFile, 
		pWriteBuff	:= ADR(I_sUeberschrift), 
		cbWriteLen	:= TO_UDINT(LEN(I_sUeberschrift)), 
		bExecute		:= TRUE, 
		tTimeout		:= T#2S, 
		bBusy			=> , 
		bError		=> , 
		nErrId		=> , 
		cbWrite		=> );
		
	IF NOT fbFileWrite.bBusy
		AND NOT fbFileWrite.bError
	THEN
		nStep:= 14;
	END_IF
///////////////////////////////////////////////////////////
14:
	fbFileWrite(
		bExecute		:= FALSE); 
	nStep:= 20;
	
///////////////////////////////////////////////////////////
20: // Schreibe Datei
	sZeile:= CONCAT(I_sZeile,'$R');
	fbFileWrite(
		sNetId		:= , 
		hFile			:= fbFileOpen.hFile, 
		pWriteBuff	:= ADR(sZeile), 
		cbWriteLen	:= TO_UDINT(LEN(sZeile)), 
		bExecute		:= TRUE, 
		tTimeout		:= T#2S, 
		bBusy			=> , 
		bError		=> , 
		nErrId		=> , 
		cbWrite		=> );
		
	IF NOT fbFileWrite.bBusy
		AND NOT fbFileWrite.bError
	THEN
		nStep:= 30;
	END_IF
	
///////////////////////////////////////////////////////////
30: // Schließe Datei
	fbFileClose(
		sNetId	:= , 
		hFile		:= fbFileOpen.hFile, 
		bExecute	:= TRUE, 
		tTimeout	:= T#2S, 
		bBusy		=> , 
		bError	=> , 
		nErrId	=> );
		
	IF NOT fbFileClose.bBusy
		AND NOT fbFileClose.bError
	THEN
		nStep:= 40;
	END_IF
	
///////////////////////////////////////////////////////////
40: // Melde DONE
	Q_bDone := TRUE;
	IF NOT I_bStart
	THEN
		nStep:= 0;
	END_IF
///////////////////////////////////////////////////////////
END_CASE

END_FUNCTION_BLOCK

// POUs/Logging/FB_TaktzeitAuswert
FUNCTION_BLOCK FB_TaktzeitAuswert
VAR_INPUT
	I_bTaktStart				: BOOL;		// Startet die Messung (z.B. Zutransport)
	I_bTaktEnde					: BOOL;		// Stoppt die Messung (z.B. Austransport beendet)
	I_bWartezeit1Start		: BOOL;		// Startet die Pausenzeitmessung (z.B. Bedienereingriff/ Warten auf Auslauffreigabe)
	I_bWartezeit1Ende			: BOOL;		// Stoppt die Pausenzeitmessung
	I_bWartezeit2Start		: BOOL;		// Startet die Pausenzeitmessung (z.B. Bedienereingriff/ Warten auf Auslauffreigabe)
	I_bWartezeit2Ende			: BOOL;		// Stoppt die Pausenzeitmessung
	I_sWartezeit1				: STRING;	// Worauf wird gewartet?
	I_sWartezeit2				: STRING;	// Worauf wird gewartet?
	I_sBearbeitung				: STRING;	// Welche Bearbeitung wird gezählt
	I_fHoehe						: LREAL;		// Teilehöhe
	I_fBreite					: LREAL;		// Teilebreite
	I_fTiefe						: LREAL;		// Teiletiefe
	I_nAnzahlBearbeitungen	: INT;		// Anzahl der Bearbeitungen am Bauteil
	
	I_bSpeicherInDatei		: BOOL;		// Wenn aktiv werden die Daten in eine Datei geschrieben
	I_sStation					: STRING;	// Stationsname
	I_sDateipfad				: STRING;	// Dateipfad ohne Dateinamen
END_VAR
VAR_OUTPUT
	Q_sUeberschrift	: T_MaxString;
	Q_sLetzteMessung	: T_MaxString;
	Q_arrTaktzeiten	: ARRAY [1..100] OF T_MaxString;
END_VAR
VAR
	rtrigTaktStart			: R_TRIG;
	rtrigTaktEnde			: R_TRIG;
	rtrigWartezeit1Start	: R_TRIG;
	rtrigWartezeit1Ende	: R_TRIG;
	rtrigWartezeit2Start	: R_TRIG;
	rtrigWartezeit2Ende	: R_TRIG;
	tonTimer	: TON;
	
	bTaktStart				: BOOL;
	bStartWartezeit1		: BOOL;
	bStartWartezeit2		: BOOL;
	
	tStartzeitTakt		: TIME;
	tEndzeitzeitTakt	: TIME;
	tStartWartezeit1	: TIME;
	tEndeWartezeit1	: TIME;
	tWartezeit1			: TIME;
	tStartWartezeit2	: TIME;
	tEndeWartezeit2	: TIME;
	tWartezeit2			: TIME;
	tTaktzeit			: TIME;
	tTaktzeitWartezeiten	: TIME;
	
	sTaktzeit				: STRING;
	sTaktzeitOhnePause	: STRING;
	sWartezeit1				: STRING:= '0';
	sWartezeit2				: STRING:= '0';
	
	sLetzterSpeicherdatensatz	: T_MaxString;
	fbLogToFile			: FB_LogToFile;
	
	fHoehe				: LREAL;
	fBreite				: LREAL;
	fTiefe				: LREAL;
	
	nIdx						: INT;
END_VAR

Q_sUeberschrift	:= '';
Q_sUeberschrift	:= CONCAT(Q_sUeberschrift,'Taktzeit[ms];Warte auf ');
Q_sUeberschrift	:= CONCAT(Q_sUeberschrift,I_sWartezeit1);
Q_sUeberschrift	:= CONCAT(Q_sUeberschrift,'[ms];Warte auf ');
Q_sUeberschrift	:= CONCAT(Q_sUeberschrift,I_sWartezeit2);
Q_sUeberschrift	:= CONCAT(Q_sUeberschrift,'[ms];Taktzeit ohne Wartezeit[ms];Höhe;Breite;Tiefe;Anzahl ');
Q_sUeberschrift	:= CONCAT(Q_sUeberschrift,I_sBearbeitung);
Q_sUeberschrift	:= CONCAT(Q_sUeberschrift,';$R');


rtrigTaktStart(CLK:= I_bTaktStart);
rtrigTaktEnde(CLK:= I_bTaktEnde);
rtrigWartezeit1Start(CLK:= I_bWartezeit1Start);
rtrigWartezeit1Ende(CLK:= I_bWartezeit1Ende);
rtrigWartezeit2Start(CLK:= I_bWartezeit2Start);
rtrigWartezeit2Ende(CLK:= I_bWartezeit2Ende);

tonTimer(IN := NOT tonTimer.Q,
			PT := t#24h);

IF rtrigTaktStart.Q
THEN
	bTaktStart				:= TRUE;
	tWartezeit1				:= T#0ms;
	sWartezeit1				:= '0';
	tWartezeit2				:= T#0ms;
	sWartezeit2				:= '0';
	tStartzeitTakt			:= tonTimer.ET;
END_IF
IF rtrigWartezeit1Start.Q
	AND bTaktStart
THEN
	bStartWartezeit1		:= TRUE;
	tStartWartezeit1		:= tonTimer.ET;
END_IF
IF rtrigWartezeit2Start.Q
	AND bTaktStart
THEN
	bStartWartezeit2		:= TRUE;
	tStartWartezeit2		:= tonTimer.ET;
END_IF

IF rtrigWartezeit1Ende.Q
	AND bStartWartezeit1
	AND bTaktStart
THEN
	tEndeWartezeit1	:= tonTimer.ET;
	tWartezeit1			:= tEndeWartezeit1 - tStartWartezeit1;
	sWartezeit1			:= TO_STRING(TO_DWORD(tWartezeit1));
	bStartWartezeit1	:= FALSE;
END_IF
IF rtrigWartezeit2Ende.Q
	AND bStartWartezeit2
	AND bTaktStart
THEN
	tEndeWartezeit2	:= tonTimer.ET;
	tWartezeit2			:= tEndeWartezeit2 - tStartWartezeit2;
	sWartezeit2			:= TO_STRING(TO_DWORD(tWartezeit2));
	bStartWartezeit2	:= FALSE;
END_IF

IF I_fHoehe <> 0
	AND bTaktStart
THEN
	fHoehe	:= I_fHoehe;
END_IF

IF I_fBreite <> 0
	AND bTaktStart
THEN
	fBreite	:= I_fBreite;
END_IF

IF I_fTiefe <> 0
	AND bTaktStart
THEN
	fTiefe	:= I_fTiefe;
END_IF


IF rtrigTaktEnde.Q
THEN
	bTaktStart				:= FALSE;
	tEndzeitzeitTakt		:= tonTimer.ET;
	tTaktzeit				:= tEndzeitzeitTakt 
									- tStartzeitTakt;
	tTaktzeitWartezeiten	:= tTaktzeit 
									- tWartezeit1 
									- tWartezeit2;
	sTaktzeit				:= TO_STRING(TO_DWORD(tTaktzeit));
	sTaktzeitOhnePause	:= TO_STRING(TO_DWORD(tTaktzeitWartezeiten));
	
	FOR nIdx := 100 TO 2 BY -1 DO
		Q_arrTaktzeiten[nIdx] := Q_arrTaktzeiten[nIdx-1];
	END_FOR
	Q_arrTaktzeiten[1]	:= '';
	Q_arrTaktzeiten[1]	:= CONCAT(Q_arrTaktzeiten[1],sTaktzeit);
	Q_arrTaktzeiten[1]	:= CONCAT(Q_arrTaktzeiten[1],';');
	Q_arrTaktzeiten[1]	:= CONCAT(Q_arrTaktzeiten[1],sWartezeit1);
	Q_arrTaktzeiten[1]	:= CONCAT(Q_arrTaktzeiten[1],';');
	Q_arrTaktzeiten[1]	:= CONCAT(Q_arrTaktzeiten[1],sWartezeit2);
	Q_arrTaktzeiten[1]	:= CONCAT(Q_arrTaktzeiten[1],';');
	Q_arrTaktzeiten[1]	:= CONCAT(Q_arrTaktzeiten[1],sTaktzeitOhnePause);
	Q_arrTaktzeiten[1]	:= CONCAT(Q_arrTaktzeiten[1],';');
	Q_arrTaktzeiten[1]	:= CONCAT(Q_arrTaktzeiten[1],TO_STRING(fHoehe));
	Q_arrTaktzeiten[1]	:= CONCAT(Q_arrTaktzeiten[1],';');
	Q_arrTaktzeiten[1]	:= CONCAT(Q_arrTaktzeiten[1],TO_STRING(fBreite));
	Q_arrTaktzeiten[1]	:= CONCAT(Q_arrTaktzeiten[1],';');
	Q_arrTaktzeiten[1]	:= CONCAT(Q_arrTaktzeiten[1],TO_STRING(fTiefe));
	Q_arrTaktzeiten[1]	:= CONCAT(Q_arrTaktzeiten[1],';');
	Q_arrTaktzeiten[1]	:= CONCAT(Q_arrTaktzeiten[1],TO_STRING(I_nAnzahlBearbeitungen));
	Q_arrTaktzeiten[1]	:= CONCAT(Q_arrTaktzeiten[1],';');
	
	Q_sLetzteMessung	:= Q_arrTaktzeiten[1];
END_IF

a_DateiSchreiben();

ACTION a_DateiSchreiben:

fbLogToFile(
	I_sDateipfad	:= I_sDateipfad, 
	I_sDateiname	:= I_sStation, 
	I_sUeberschrift:= Q_sUeberschrift, 
	I_sZeile			:= Q_sLetzteMessung);
	
IF Q_sLetzteMessung <> sLetzterSpeicherdatensatz
	AND Q_sLetzteMessung <> '0;0;0;0;0.0;0.0;0.0;0;'
	AND I_bSpeicherInDatei
THEN
	fbLogToFile(
		I_bStart			:= TRUE);
END_IF

IF fbLogToFile.Q_bDone
THEN
	fbLogToFile(
		I_bStart	:= FALSE);
	sLetzterSpeicherdatensatz 	:= Q_sLetzteMessung;
END_IF
END_ACTION

END_FUNCTION_BLOCK

// POUs/MeldTest/FB_MeldTestAllgemein
// Dies ist ein Testbaustein, um alle Standardmeldunge, die in der Bibliothek vordefiniert sind, auszulösen.
// Sie werden im Anschluss nicht zurückgesetzt!
FUNCTION_BLOCK FB_MeldTestAllgemein
VAR_IN_OUT
	st0100Meldungen 	: ST_0100_Meldungen;
END_VAR
VAR
	nIdx	: INT;
END_VAR

For nIdx := 1 TO cAnzKlimageraete DO
	st0100Meldungen.stSchaltSchr.arrMeldKlimageraet[nIdx].bMeldAusg 				:= TRUE;
END_FOR
For nIdx := 1 TO cAnzNetzteile DO
	st0100Meldungen.stSchaltSchr.arrMeldNetzteil[nIdx].bMeldAusg 					:= TRUE;
END_FOR
For nIdx := 1 TO cAnzSicherungen DO
	st0100Meldungen.stSchaltSchr.arrMeldSicherung[nIdx].bMeldAusg 					:= TRUE;
END_FOR
For nIdx := 1 TO cAnzElekSicherungen DO
	st0100Meldungen.stSchaltSchr.arrMeldElektSicherung[nIdx].bMeldAusg 			:= TRUE;
END_FOR
For nIdx := 1 TO cAnzMSSchalter DO
	st0100Meldungen.stSchaltSchr.arrMeldMotorschutz[nIdx].bMeldAusg 				:= TRUE;
END_FOR
For nIdx := 1 TO cAnzThermoueberw DO
	st0100Meldungen.stSchaltSchr.arrMeldThermoueberw[nIdx].bMeldAusg				:= TRUE;
END_FOR
For nIdx := 1 TO cAnzWartungsEinheit DO
	st0100Meldungen.stSchaltSchr.arrBetriebsdruck[nIdx].bMeldBetriebsdruck 		:= TRUE;
END_FOR
st0100Meldungen.stSchaltSchr.stMeldAusgUSV.bMeldAustausch				 			:= 
st0100Meldungen.stSchaltSchr.stMeldAusgUSV.bMeldBatteriebetrieb		 			:= 
st0100Meldungen.stSchaltSchr.stMeldAusgUSV.bMeldKommFehler				 			:= 
st0100Meldungen.stSchaltSchr.stMeldAusgUSV.bMeldKritLevel				 			:= 
st0100Meldungen.stSchaltSchr.stMeldAusgUSV.bMeldStatusUnbekannt		 			:= 
st0100Meldungen.stSchaltSchr.stMeldAusgUSV.bMeldUnteresLevel			 			:= TRUE;

For nIdx := 1 TO cAnzEinspeis DO
	st0100Meldungen.stEinspeis.arrMeldEinspeis[nIdx].bMeldRueckspeis 				:= 
	st0100Meldungen.stEinspeis.arrMeldEinspeis[nIdx].bMeldEinspeis	 				:= TRUE;
END_FOR
For nIdx := 1 TO cAnzAuffrisch DO
	st0100Meldungen.stEinspeis.arrMeldAuffrisch[nIdx].bMeldUnterspannung 		:= TRUE;
END_FOR
FOR nIdx := 1 TO cAnzKommError DO
	st0100Meldungen.stKommunikation.arrMeldKommError[nIdx].bMeldKommError		:= TRUE; 
END_FOR
FOR nIdx := 1 TO cAnzADS_EA_Error DO
	st0100Meldungen.stKommunikation.arrMeldADS_EA_Error[nIdx].bError				:= TRUE; 
END_FOR
FOR nIdx := 1 TO cAnzADS_Data_Error DO
	st0100Meldungen.stKommunikation.arrMeldADS_Data_Error[nIdx].bError	 		:= TRUE; 
END_FOR

FOR nIdx := 1 TO cAnzWartungstuer DO
	st0100Meldungen.stSchutzbereiche.arrMeldWartgTuer[nIdx].bMeldGeoeffnet		:= 
	st0100Meldungen.stSchutzbereiche.arrMeldWartgTuer[nIdx].bMeldAutoHalt		:= TRUE; 	
END_FOR
FOR nIdx := 1 TO cAnzLichtgitter DO
	st0100Meldungen.stSchutzbereiche.arrMeldSichLichtg[nIdx].bMeldAusg			:= TRUE; 	
END_FOR
FOR nIdx := 1 TO cAnzNotHalt DO
	st0100Meldungen.stSchutzbereiche.arrMeldNotHalt[nIdx].bMeldAusg				:= TRUE; 	
END_FOR
FOR nIdx := 1 TO cAnzSchutzBer DO
	st0100Meldungen.stSchutzbereiche.arrMeldStHLuft[nIdx].bMeldNichtAbgebaut				:=
	st0100Meldungen.stSchutzbereiche.arrMeldStHLuft[nIdx].bMeldNichtAufgebaut				:=
	st0100Meldungen.stSchutzbereiche.arrMeldStHLuft[nIdx].bMeldNichtFreigegeben			:=
	st0100Meldungen.stSchutzbereiche.arrMeldTuerFrgBremsentest[nIdx].bMeldGesperrt		:=
	st0100Meldungen.stSchutzbereiche.arrMeldSchutzbereichOffen[nIdx].bMeldUnterbrochen	:= TRUE; 	
END_FOR

FOR nIdx := 1 TO cAnzAchsGruppen DO
	st0100Meldungen.stAchsen.stMeldAchsfehler.bMeldFreifahren									:= 
	st0100Meldungen.stAchsen.stMeldAchsfehler.bMeldReset											:= 
	st0100Meldungen.stAchsen.arrMeldAchsGruppe[nIdx].bMeldFehler								:= TRUE; 	
END_FOR

	st0100Meldungen.stDatenanf.bMeldAnfFehler															:= 
	st0100Meldungen.stEtherCAT.bMeldAnzSlavesFehler													:= 
	st0100Meldungen.stEtherCAT.bMeldEtherCATFehler													:= 
	st0100Meldungen.stEtherCAT.bMeldSlaveError														:= TRUE;

FOR nIdx := 1 TO cAnzSafetyGruppen DO
	st0100Meldungen.stSafety.arrMeldGruppen[nIdx].bMeldAusg										:=
	st0100Meldungen.stSafety.arrMeldGruppen[nIdx].bMeldFBErrorGrp								:=  TRUE; 	
END_FOR
FOR nIdx := 1 TO cAnzSafetyFBError DO
	st0100Meldungen.stSafety.arrMeldFBErrors[nIdx].bMeldFBError_ErrorDiag					:=
	st0100Meldungen.stSafety.arrMeldFBErrors[nIdx].bMeldFBError_ErrorState					:=  TRUE; 	
END_FOR

END_FUNCTION_BLOCK

// POUs/Time/FB_Zeitstempel
// Mit diesem FB wird zentral die aktuelle Systemzeit ermittelt und in die Strukturen ST_TimeStamp und ST_TimeStrukt geschrieben.
// in der ST_TimeStamp wird die Systemzeit einmal in der Sekunde als String generiert.
// zusätzlich werden die globalen Variablen stTimestamp und stTimestruct beschrieben.
// Dieser FB solle im Main-Programm aufgerufen werden.
FUNCTION_BLOCK FB_Zeitstempel
VAR_INPUT
	I_bHochkomma 		: BOOL;					// Jeweils Datum und Uhrzeit in Hochkommata. Wenn FALSE dann ohne "
	I_bSemikolon		: BOOL;					// Datum- Uhrzeit-Treuung mit Semikolon. Wenn FALSE dann mit  Bindestrich
	I_CycleTime			: UDINT;					// Obsolet. Das wird jetzt über einen internen Time gelöst
END_VAR
VAR_OUTPUT
	Q_stTimestamp	:	ST_TimeStamp;			// Alle Ausgangswerte zusammengefasst
	Q_stTimestruct	:	ST_TimeStruct;			// Alle Ausgangswerte um einen String mit allen Werten erweitert
END_VAR
VAR
	bInitOk			:	BOOL;						// Für einmaliges Lesen der Zykluszeit
	nSPS_Taskzeit	:	UINT;						// Ermittelte SPS-Zykluszeit
	sQ1				:	STRING;					// Hilfvariable zur Formaterzeugung
	
	tonUpdate		: TON;						// Timer um einmal in der Sekunde den String im Timstamp zu aktualisieren

	sHochkomma		:	STRING(2);				// Hochkomma-Platzhalter
	sSemikolon		:	STRING(3);				// Semikolon-Platzhalter
	stTimeStr		:	Tc2_Utilities.TIMESTRUCT;	// Struktur zum Lesen der Zeit
	fbgettime		:	Tc2_Utilities.NT_GetTime;	// Instanz zum Lesen der Windows-Zeit
END_VAR

//****************************************************************************************************

	IF I_bHochkomma
	THEN
		sHochkomma := '"';
	ELSE
		sHochkomma := '';
	END_IF

	IF I_bSemikolon
	THEN
		sSemikolon := ';';
	ELSE
		sSemikolon := ' - ';
	END_IF
	
	// GET-Time zyklisch aufrufen, damit auch die Millisekunden erfasst werden.
	fbgettime(START := NOT fbgettime.BUSY);
	fbgettime(START := FALSE);

	Q_stTimestamp.nMilliSekunde	:= fbgettime.TIMESTR.wMilliseconds;
	
	tonUpdate(
		IN	:= NOT tonUpdate.Q,
		PT	:= T#1s
	);
	
//****************************************************************************************************
	// TimeStruct nur einmal in der Sekunde beschreiben
	IF	tonUpdate.Q
	THEN

		(* Zeitstring holen *)
		stTimeStr := fbgettime.TIMESTR;

		sQ1 := '';

		(* ggf Hochkomma wenn CSV-Datei *)
		sQ1 := CONCAT(sQ1,sHochkomma);

		//****************************************************************************************************
		(* Tag *)
		IF stTimeStr.wDay < 10
		THEN
			sQ1 := CONCAT(sQ1,'0');
		END_IF
		sQ1 := CONCAT(sQ1,WORD_TO_STRING(stTimeStr.wDay));
		sQ1 := CONCAT(sQ1,'.');

		Q_stTimestamp.nTag				:=	stTimeStr.wDay;
		Q_stTimestamp.nTagDerWoche	:=	stTimeStr.wDayOfWeek;

		//****************************************************************************************************
		(* Monat *)
		IF stTimeStr.wMonth < 10
		THEN
			sQ1 := CONCAT(sQ1,'0');
		END_IF
		sQ1 := CONCAT(sQ1,WORD_TO_STRING(stTimeStr.wMonth));
		sQ1 := CONCAT(sQ1,'.');

		Q_stTimestamp.nMonat	:=	stTimeStr.wMonth;

		//****************************************************************************************************
		(* Jahr *)
		sQ1 := CONCAT(sQ1,WORD_TO_STRING(stTimeStr.wYear));

		Q_stTimestamp.nJahr	:=	stTimeStr.wYear;

		//****************************************************************************************************
		(* ggf Hochkomma wenn CSV-Datei *)
		sQ1 := CONCAT(sQ1,sHochkomma);

		//****************************************************************************************************
		(* Trennung *)
		sQ1 := CONCAT(sQ1,sSemikolon);

		(* ggf Hochkomma wenn CSV-Datei *)
		sQ1 := CONCAT(sQ1,sHochkomma);

		//****************************************************************************************************
		(* Stunde *)
		IF stTimeStr.wHour < 10
		THEN
			sQ1 := CONCAT(sQ1,'0');
		END_IF

		sQ1 := CONCAT(sQ1,WORD_TO_STRING(stTimeStr.wHour));
		sQ1 := CONCAT(sQ1,':');

		Q_stTimestamp.nStunde	:=	stTimeStr.wHour;

		//****************************************************************************************************
		(* Minute *)
		IF stTimeStr.wMinute < 10
		THEN
			sQ1 := CONCAT(sQ1,'0');
		END_IF

		sQ1 := CONCAT(sQ1,WORD_TO_STRING(stTimeStr.wMinute));
		sQ1 := CONCAT(sQ1,':');

		Q_stTimestamp.nMinute	:=	stTimeStr.wMinute;

		//****************************************************************************************************
		(* Sekunde *)
		IF stTimeStr.wSecond < 10
		THEN
			sQ1 := CONCAT(sQ1,'0');
		END_IF

		sQ1 := CONCAT(sQ1,WORD_TO_STRING(stTimeStr.wSecond));
		sQ1 := CONCAT(sQ1,':');

		Q_stTimestamp.nSekunde	:=	stTimeStr.wSecond;
	
	END_IF
	
	//****************************************************************************************************
	(* Millisekunde *)
	// Dieser Bereich wird zyklisch geupdated
	
	IF (fbgettime.TIMESTR.wMilliseconds < 100)
		AND (fbgettime.TIMESTR.wMilliseconds > 9)
	THEN
		Q_stTimestamp.sQ := CONCAT('0', WORD_TO_STRING(fbgettime.TIMESTR.wMilliseconds));
	ELSIF fbgettime.TIMESTR.wMilliseconds < 10
	THEN
		Q_stTimestamp.sQ := CONCAT('00', WORD_TO_STRING(fbgettime.TIMESTR.wMilliseconds));
	ELSE
		Q_stTimestamp.sQ := WORD_TO_STRING(fbgettime.TIMESTR.wMilliseconds);
	END_IF

	// Millisekunden an den TimeStamp ergänzen
	IF LEN(sQ1) > 0
	THEN
		Q_stTimestamp.sQ := CONCAT(sQ1,Q_stTimestamp.sQ);

		// ggf Hochkomma wenn CSV-Datei
		Q_stTimestamp.sQ := CONCAT(Q_stTimestamp.sQ,sHochkomma);

	END_IF
	
//****************************************************************************************************
// Hier wird der originale TimeStruct um seinen String erweitert.
	IF I_bSemikolon
	THEN
		Q_stTimestruct:= F_TimeStruct(fbgettime.TIMESTR,';');
	ELSE
		Q_stTimestruct:= F_TimeStruct(fbgettime.TIMESTR,'-');
	END_IF

//****************************************************************************************************
// Werte in globale Lib-Variabelen schreiben
	GlobalVar_Allgemein.stTimestamp 	:= Q_stTimestamp;
	GlobalVar_Allgemein.stTimestruct	:= Q_stTimestruct;
	
//****************************************************************************************************
// ENDE

END_FUNCTION_BLOCK

// POUs/UniBausteine/FB_LaufzMeldg
// Funktionsbaustein zur Überwachung der Ein- und Ausgangszustände von dem UniZyliAnstg-Baustein.
FUNCTION_BLOCK FB_LaufzMeldg
VAR_INPUT

	I_bLaufzAnstg0		:BOOL;	// Zu überwachender Ausgang für Ventil Richtung 0-Position schalten
	I_bLaufzAbfrg0		:BOOL;	// Hardware-Eingang, Zylinder ist in 0-Position
	I_bLaufzAnstg1		:BOOL;	// Zu überwachender Ausgang für Ventil Richtung 1-Position schalten
	I_bLaufzAbfrg1		:BOOL;	// Hardware-Eingang, Zylinder ist in 1-Position

	I_bMeldgFreig		:BOOL;	// Ablauf der Laufzeitmeldung wird freigegeben. Erst wenn TRUE läuft die Zeit ab.

	I_tLaufzDauer		:TIME;	// Laufzeit bis die Meldungen kommen

END_VAR
VAR_OUTPUT

	Q_bLaufzMeldg0		:BOOL;	// Laufzeit für Zylinder ist nicht in 0-Position
	Q_bLaufzMeldg1		:BOOL;	// Laufzeit für Zylinder ist nicht in 1-Position
	Q_bSensMeldg		:BOOL;	// Beide Sensoren sind an.

END_VAR
VAR
	tonVerzMeldg0		:TON;
	tonVerzMeldg1		:TON;
END_VAR

	(*Allg.- Laufzeitmeldung*)

	tonVerzMeldg0 (IN:= I_bLaufzAnstg0 
				AND NOT I_bLaufzAbfrg0 
				AND I_bMeldgFreig, 
				PT:= I_tLaufzDauer);
				
	IF tonVerzMeldg0.Q
	THEN
		Q_bLaufzMeldg0:= TRUE;
	ELSIF I_bLaufzAbfrg0
		OR I_bLaufzAnstg1
		OR NOT I_bMeldgFreig
	THEN
		Q_bLaufzMeldg0:= FALSE;
	END_IF

	tonVerzMeldg1 (IN:= I_bLaufzAnstg1 
				AND NOT I_bLaufzAbfrg1 
				AND I_bMeldgFreig, 
				PT:= I_tLaufzDauer);	

	IF tonVerzMeldg1.Q
	THEN
		Q_bLaufzMeldg1:= TRUE;
	ELSIF I_bLaufzAbfrg1
		OR I_bLaufzAnstg0
		OR NOT I_bMeldgFreig
	THEN
		Q_bLaufzMeldg1:= FALSE;
	END_IF

	Q_bSensMeldg:= I_bLaufzAbfrg0 
				AND I_bLaufzAbfrg1 
				AND I_bMeldgFreig;

// ENDE

END_FUNCTION_BLOCK

// POUs/UniBausteine/FB_LaufzMeldgAktr
// Funktionsbaustein zur Überwachung der Ein- und Ausgangszustände von dem UniZyliAnstg-Baustein.
FUNCTION_BLOCK FB_LaufzMeldgAktr
VAR_INPUT

	I_bLaufzAnstg0		:BOOL;	// Zu überwachender Ausgang für Ventil Richtung 0-Position schalten
	I_bLaufzAbfrg0		:BOOL;	// Hardware-Eingang, Zylinder ist in 0-Position
	I_bLaufzAnstg1		:BOOL;	// Zu überwachender Ausgang für Ventil Richtung 1-Position schalten
	I_bLaufzAbfrg1		:BOOL;	// Hardware-Eingang, Zylinder ist in 1-Position

	I_bMeldgFreig		:BOOL;	// Ablauf der Laufzeitmeldung wird freigegeben. Erst wenn TRUE läuft die Zeit ab.

	I_tLaufzDauer		:TIME;	// Laufzeit bis die Meldungen kommen

END_VAR
VAR_OUTPUT

	Q_bLaufzMeldg0		:BOOL;	// Laufzeit für Zylinder ist nicht in 0-Position
	Q_bLaufzMeldg1		:BOOL;	// Laufzeit für Zylinder ist nicht in 1-Position
	Q_bSensMeldg		:BOOL;	// Beide Sensoren sind an.

END_VAR
VAR
	tonVerzMeldg0		:TON;
	tonVerzMeldg1		:TON;
END_VAR

	(*Allg.- Laufzeitmeldung*)

	tonVerzMeldg0 (IN:= I_bLaufzAnstg0 
				AND NOT I_bLaufzAbfrg0 
				AND I_bMeldgFreig, 
				PT:= I_tLaufzDauer);
				
	IF tonVerzMeldg0.Q
	THEN
		Q_bLaufzMeldg0:= TRUE;
	ELSIF I_bLaufzAbfrg0
		OR I_bLaufzAnstg1
		OR NOT I_bLaufzAnstg0
		OR NOT I_bMeldgFreig
	THEN
		Q_bLaufzMeldg0:= FALSE;
	END_IF

	tonVerzMeldg1 (IN:= I_bLaufzAnstg1 
				AND NOT I_bLaufzAbfrg1 
				AND I_bMeldgFreig, 
				PT:= I_tLaufzDauer);	

	IF tonVerzMeldg1.Q
	THEN
		Q_bLaufzMeldg1:= TRUE;
	ELSIF I_bLaufzAbfrg1
		OR I_bLaufzAnstg0
		OR NOT I_bLaufzAnstg1
		OR NOT I_bMeldgFreig
	THEN
		Q_bLaufzMeldg1:= FALSE;
	END_IF

	Q_bSensMeldg:= I_bLaufzAbfrg0 
				AND I_bLaufzAbfrg1 
				AND I_bMeldgFreig;

// ENDE

END_FUNCTION_BLOCK

// POUs/UniBausteine/FB_UniAchsAnstg
(*
Beschreibung :	UniFB zur Handsteuerung, Anzeige und Fehlermeldungen in der Avalon-HMI einer NC-Achse als Servo bzw. Sercos-Achse.
					Die Kommunikation mit der NC erfolgt über IQ_stAchse und die eigentliche Steuerung über FB_AchsKontrlAnstg.
					inkl. Handling - Handfunktinen
										- Meldefunktionen
										- Betriebsarten
										- Schutzbereiche
					Datentypen: ST_UniBaustein
									ST_UniAchsAnstg
									ST_NcAchsen
					Ressourcen: GlobalVar_Allgemein
									GlobalVar_Farben
									AllgemeineParameter
TwinCat Vers.:	3.1.4024.25							
Erstellt		 :	Anlagentechnik Grp.11 (BECKHOFF AUTOMATION)
*)
FUNCTION_BLOCK FB_UniAchsAnstg
VAR_INPUT

	I_sSchaltSchr		:Tc2_System.T_MaxString;	(*Aktueller Schaltschrank in dem der Regler sitzt.*)
	I_sAktorName		:Tc2_System.T_MaxString;	(*Aktueller Aktorname*)
	I_sAchsnummer		:Tc2_System.T_MaxString;	(*Aktuelle Achsnummer (Hüttenhölscher-Achsnummer)*)
	I_sAktorBMK			:Tc2_System.T_MaxString;	(*BMK - Betriebsbereit*)
	I_sEndlgBMK0		:Tc2_System.T_MaxString;	(*BMK - negative Endlage*)
	I_sEndlgBMK1		:Tc2_System.T_MaxString;	(*BMK - positive Endlage*)
	
	I_bAbfrStatUmr		:BOOL;	(*Statusabfrage Umrichter*)
																															
	I_nSchutzBer		:INT;		(*Schutzbereich => Betriebsart*)

	// Optionale Funktionen													
	I_bVerrHdFktP		:BOOL;	(*Sperren Handfkt. Pos. Richtg.*)	
	I_bVerrHdFktN		:BOOL;	(*Sperren Handfkt. Neg. Richtg.*)

END_VAR
VAR_IN_OUT
																							
	IQ_stUniAnstgHMI	:ST_UniAchsAnstg;	// HMI-Strukturen
	IQ_stAchse			:ST_NcAchsen;	// arrNcAchsen[xy] muss hier angelegt werden.

END_VAR
VAR

	bHdFktReset			:BOOL;												
	bHdUmrMeldg			:BOOL;
	
	tonMeldNichtBtb	:TON;

	//Relevante Variablen zur Diagnose
	stUniAnstgFkt		:ST_UniBaustein;

END_VAR

	(*Uni.- Achsenansteuerung*)
	
	(**************************************************)	
	(*Aufruf-Bereichskontrolle*)

	IF I_nSchutzBer <= 0 OR I_nSchutzBer > cAnzSchutzBer
		THEN
			IQ_stUniAnstgHMI.stMeldAusgHMI.sMeldText		:= 'I_nSchutzBer = 0 oder zu gross.';

			IQ_stUniAnstgHMI.stMeldAusgHMI.SourceName		:= I_sSchaltSchr;
			IQ_stUniAnstgHMI.stMeldAusgHMI.sInfoText		:= I_sAktorName;
		 	IQ_stUniAnstgHMI.stMeldAusgHMI.sBMK				:= I_sAktorBMK;
		 	IQ_stUniAnstgHMI.stMeldAusgHMI.sAchsnummer	:= I_sAchsnummer;
					
			IQ_stUniAnstgHMI.stMeldAusgHMI.bMeldHinweis	:= TRUE;
			stUniAnstgFkt.nHandStat:= 256;	// Funktion sperren
			
			y_ZustAnzg();
			RETURN;
		ELSE
			IQ_stUniAnstgHMI.stMeldAusgHMI.bMeldHinweis	:= FALSE;
			IQ_stUniAnstgHMI.stMeldAusgHMI.sMeldText		:= '';
	END_IF

	(**************************************************)	
	(*Haendling Uni-Struktur*)

	a_Standard();

	(**************************************************)	
	(*Signale austauschen*)

	w_InOutNc();
	
	(**************************************************)	
	(*Zustände anzeigen*)

	y_ZustAnzg();

	(**************************************************)	
	(*Meldungen ausgeben*)

	z_FehlMeld();
	
	(**************************************************)

ACTION a_Standard:
	(*Ansteuerungstyp "Standard" /z.B. Servoantriebe...*)

	(*Verwendete Softkeytasten = 5 (s.Beispiel)*)

   (*       "Handfunktion"       /   "Softkeytaste 1"   /   "Softkeytaste 2"   /   "Softkeytaste 3"   /   "Softkeytaste 4"   /   "Softkeytaste 5"   *)
	(*                                                                          															  								 *) 
	(*----- X-Aggregatachse ------/____negativ fahren____/____positiv fahren____/_________Frei_________/_________Frei_________/________Reset_________*)
	
	(*Softkeyleiste.1		:Funktion Tastend aktiv /Richtg. Negativ*)
	(*Softkeyleiste.2		:Funktion Tastend aktiv /Richtg. Positiv*)
	(*Softkeyleiste.3		:Platzhalter				 					 *)
	(*Softkeyleiste.4		:Platzhalter				 					 *)
	(*Softkeyleiste.5		:Funktion Umrichter-Reset					 *)

	(*Hinweis:
	- Funktion wird durch "VerrHdFkt" gesperrt (z.B. bei Kollissionserkennung...)
	*)

	(**************************************************)	

	stUniAnstgFkt.bHandAnw0:= IQ_stUniAnstgHMI.stHandFktHMI[1].bySwitch > 0;
	stUniAnstgFkt.bHandAnw1:= IQ_stUniAnstgHMI.stHandFktHMI[2].bySwitch > 0;

	bHdFktReset				  := IQ_stUniAnstgHMI.stHandFktHMI[5].bySwitch > 0;	
	
	IF arrBetrartAutomAktiv[I_nSchutzBer]
		THEN
			stUniAnstgFkt.arrHandFkt[0]:=
			stUniAnstgFkt.arrHandFkt[1]:= FALSE;
		ELSE
			IF NOT arrBetrartAutomSpeichn[I_nSchutzBer] THEN
				IF NOT arrGrdstlgBetrAktiv[I_nSchutzBer] THEN
					stUniAnstgFkt.arrHandFkt[1]:= arrBetrartHandAktiv[I_nSchutzBer]
													  		AND stUniAnstgFkt.bHandAnw1
													  		AND NOT stUniAnstgFkt.bHandAnw0
													  		AND NOT I_bVerrHdFktP	
													  		AND IQ_stAchse.stFreigb.bVorsFrgPos;
					stUniAnstgFkt.arrHandFkt[0]:= arrBetrartHandAktiv[I_nSchutzBer]
													  		AND stUniAnstgFkt.bHandAnw0
													  		AND NOT stUniAnstgFkt.bHandAnw1
													  		AND NOT I_bVerrHdFktN
													  		AND IQ_stAchse.stFreigb.bVorsFrgNeg;
				END_IF
			END_IF
	END_IF

	IF arrBetrartHandAktiv[I_nSchutzBer]
		THEN
			stUniAnstgFkt.nHandStat:= 0;			(*Funktion freigegeben*)
			IF stUniAnstgFkt.arrHandFkt[1]
				THEN
					stUniAnstgFkt.nHandStat:= 2;	(*Handfunktion.2 aktiv*)
			END_IF
			IF stUniAnstgFkt.arrHandFkt[0]
				THEN
					stUniAnstgFkt.nHandStat:= 1;	(*Handfunktion.1 aktiv*)
			END_IF
		ELSE
			stUniAnstgFkt.nHandStat:= 256;		(*Funktion gesperrt*)
	END_IF

	(**************************************************)	
	
	IQ_stAchse.stGrdfkt.bHdfkt_pos:=	stUniAnstgFkt.arrHandFkt[1];
	IQ_stAchse.stGrdfkt.bHdfkt_neg:=	stUniAnstgFkt.arrHandFkt[0];

	(**************************************************)
END_ACTION

ACTION w_InOutNc:

	(**************************************************)	
	(*Signale austauschen*)

	(*NcAchse <> Antrieb*)

	IQ_stAchse.stStatus.bAchseBTB:= I_bAbfrStatUmr;	//Umrichter-Status
	
	bHdUmrMeldg:= NOT IQ_stAchse.stStatus.bAchseBTB
				  	  AND arrAntrGruppeFrg[I_nSchutzBer];
	
//CFR	arrNcAchsenUmrReset[I_nAchsBezNr]:= bHdFktReset;	//Umrichter-Reset
	
	(**************************************************)
END_ACTION

ACTION y_ZustAnzg:
	
	(**************************************************)	
	(*Zustände anzeigen*)

	IF stUniAnstgFkt.nHandStat = 1	(*Handfunktion.1 aktiv*)
		THEN
			IQ_stUniAnstgHMI.stHandFktHMI[1].sColour:= cGruenAsString;
			IQ_stUniAnstgHMI.stHandFktHMI[1].sText:= 'negativ fahren';
		ELSE
			IQ_stUniAnstgHMI.stHandFktHMI[1].sColour:= cDefaultAsString;
			IQ_stUniAnstgHMI.stHandFktHMI[1].sText:= 'negativ fahren';
   END_IF
	IF stUniAnstgFkt.nHandStat = 2	(*Handfunktion.2 aktiv*)
		THEN		 
			IQ_stUniAnstgHMI.stHandFktHMI[2].sColour:= cGruenAsString;
			IQ_stUniAnstgHMI.stHandFktHMI[2].sText:= 'positiv fahren';
		ELSE
			IQ_stUniAnstgHMI.stHandFktHMI[2].sColour:= cDefaultAsString;
			IQ_stUniAnstgHMI.stHandFktHMI[2].sText:= 'positiv fahren';
   END_IF
	
	// In Taste 3 einfach mal die Istposition anzeigen
	IQ_stUniAnstgHMI.stHandFktHMI[3].sColour:= cDefaultAsString;
	IQ_stUniAnstgHMI.stHandFktHMI[3].sText:= CONCAT('Istposition: ', Tc2_Utilities.LREAL_TO_FMTSTR(IQ_stAchse.fPosIstwert,2,TRUE));
	IQ_stUniAnstgHMI.stHandFktHMI[4].sColour:= cDefaultAsString;
	IQ_stUniAnstgHMI.stHandFktHMI[4].sText:= CONCAT('letzte Sollposition: ', Tc2_Utilities.LREAL_TO_FMTSTR(IQ_stAchse.stAuftrg.fPTP_LetzZiel ,2,TRUE));
	
	IF bHdUmrMeldg
		THEN
			IQ_stUniAnstgHMI.stHandFktHMI[5].sColour:= cOrangeAsString;
			IQ_stUniAnstgHMI.stHandFktHMI[5].sText:= 'Reset';
		ELSE
			IQ_stUniAnstgHMI.stHandFktHMI[5].sColour:= cBlauAsString;
			IQ_stUniAnstgHMI.stHandFktHMI[5].sText:= 'Reset';
   END_IF
	IF stUniAnstgFkt.nHandStat = 256	(*Funktion gesperrt*)
		THEN
			IQ_stUniAnstgHMI.stHandFktHMI[1].byStatus:=
			IQ_stUniAnstgHMI.stHandFktHMI[2].byStatus:=
			IQ_stUniAnstgHMI.stHandFktHMI[3].byStatus:=
			IQ_stUniAnstgHMI.stHandFktHMI[4].byStatus:=
			IQ_stUniAnstgHMI.stHandFktHMI[5].byStatus:= 1;
		ELSE
			IQ_stUniAnstgHMI.stHandFktHMI[1].byStatus.0	:= I_bVerrHdFktN;
			IQ_stUniAnstgHMI.stHandFktHMI[2].byStatus.0	:= I_bVerrHdFktP;
			IQ_stUniAnstgHMI.stHandFktHMI[3].byStatus:=
			IQ_stUniAnstgHMI.stHandFktHMI[4].byStatus:=
			IQ_stUniAnstgHMI.stHandFktHMI[5].byStatus:=  0;
   END_IF
	
	(**************************************************)
END_ACTION

ACTION z_FehlMeld:

	(**************************************************)	
	(*Meldungen ausgeben*)

	IQ_stUniAnstgHMI.stMeldAusgHMI.SourceID			:= 0;	// Nicht mehr verwendet
	IQ_stUniAnstgHMI.stMeldAusgHMI.SourceName			:= I_sSchaltSchr;
	IQ_stUniAnstgHMI.stMeldAusgHMI.sInfoText			:= I_sAktorName;
	IQ_stUniAnstgHMI.stMeldAusgHMI.sAktorName			:= I_sAktorName;
 	IQ_stUniAnstgHMI.stMeldAusgHMI.sBMK					:= I_sAktorBMK;
	IQ_stUniAnstgHMI.stMeldAusgHMI.sAchsnummer		:= I_sAchsnummer;

	tonMeldNichtBtb(
		IN :=arrAntrGruppeFrg[I_nSchutzBer]
				AND NOT I_bAbfrStatUmr
				AND bVersEingAusgSchaltsOk,
		PT :=t#3s);

	IQ_stUniAnstgHMI.stMeldAusgHMI.bStatMeldAusg		:= tonMeldNichtBtb.Q;

	(**************************************************)	
	(*Zus. Meldungen Achsansteuerung*)

	IQ_stUniAnstgHMI.stAchsMeldHMI.SourceID			:= 0;	// Nicht mehr verwendet
	IQ_stUniAnstgHMI.stAchsMeldHMI.SourceName			:= I_sSchaltSchr;	
	IQ_stUniAnstgHMI.stAchsMeldHMI.sAktorIdNr			:= I_sAchsnummer;
	IQ_stUniAnstgHMI.stAchsMeldHMI.sAktorName			:= I_sAktorName;
	IQ_stUniAnstgHMI.stAchsMeldHMI.sEndlgBMK0			:= I_sEndlgBMK0;
	IQ_stUniAnstgHMI.stAchsMeldHMI.sEndlgBMK1			:= I_sEndlgBMK1;
 	IQ_stUniAnstgHMI.stAchsMeldHMI.sBMK					:= I_sAktorBMK;



	IQ_stUniAnstgHMI.stAchsMeldHMI.bMeldNCFehler				:= IQ_stAchse.bNcFehler
																				OR bTestMeldAchs;
	IQ_stUniAnstgHMI.stAchsMeldHMI.bMeldNichtBtB				:= IQ_stAchse.stMeldg.bAntrbFehl
																				OR bTestMeldAchs;
	// Hier zum BMK noch die Ist-Position hinzufügen. Die Ist-Position wünschte sich nobilia. Das BMK bietet sich dafür an. Weitere Variablen in die Meldestruktur ist nicht möglich.
	IF IQ_stAchse.stMeldg.bIstPosFehl
		OR bTestMeldAchsIstPosFehler
	THEN
		IQ_stUniAnstgHMI.stAchsMeldHMI.sBMK :=
			CONCAT(I_sAktorBMK,
			CONCAT(' Istposition: ',TO_STRING(IQ_stAchse.fPosIstwert)));
	END_IF

	IQ_stUniAnstgHMI.stAchsMeldHMI.bMeldIstPosUngueltig	:= IQ_stAchse.stMeldg.bIstPosFehl
																				OR bTestMeldAchs
																				OR bTestMeldAchsIstPosFehler;

	// Hier zum BMK noch die Soll-Position hinzufügen. Die Soll-Position wünschte sich nobilia. Das BMK bietet sich dafür an. Weitere Variablen in die Meldestruktur ist nicht möglich.
	// Dazu noch die Softwareendlagen, damit man auch weiß wohin man maximal darf.
	IF IQ_stAchse.stMeldg.bZielPosFehl
		OR bTestMeldAchs
	THEN
		IQ_stUniAnstgHMI.stAchsMeldHMI.sBMK :=
			CONCAT(I_sAktorBMK,
			CONCAT(' Zielposition: ',
			CONCAT(TO_STRING(IQ_stAchse.stAuftrg.fPTP_ZielPos),
			CONCAT(' Softwareendlage minimum: ',
			CONCAT(TO_STRING(IQ_stAchse.stParam.fSoftEndlMin),
			CONCAT(' Softwareendlage maximum: ',TO_STRING(IQ_stAchse.stParam.fSoftEndlMax)))))));
	END_IF
	
	IQ_stUniAnstgHMI.stAchsMeldHMI.bMeldZielPosUngueltig	:= IQ_stAchse.stMeldg.bZielPosFehl
																				OR bTestMeldAchs;

	// Hier zum BMK noch die Soll-Position hinzufügen. Die Soll-Position wünschte sich nobilia. Das BMK bietet sich dafür an. Weitere Variablen in die Meldestruktur ist nicht möglich.
	IF IQ_stAchse.stMeldg.bLfZeitFehl
		OR bTestMeldAchs
	THEN
		IQ_stUniAnstgHMI.stAchsMeldHMI.sBMK :=
			CONCAT(I_sAktorBMK,
			CONCAT(' Zielposition: ',TO_STRING(IQ_stAchse.stAuftrg.fPTP_ZielPos)));
	END_IF
	
	IQ_stUniAnstgHMI.stAchsMeldHMI.bMeldLaufzeitfehler		:= IQ_stAchse.stMeldg.bLfZeitFehl
																				OR bTestMeldAchs;

	// Hier zum BMK noch die Ist-Position hinzufügen. Die Ist-Position wünschte sich nobilia. Das BMK bietet sich dafür an. Weitere Variablen in die Meldestruktur ist nicht möglich.
	IF IQ_stAchse.stMeldg.bEndlNegAngf
		OR bTestMeldAchs
	THEN
		IQ_stUniAnstgHMI.stAchsMeldHMI.sBMK :=
			CONCAT(I_sAktorBMK,
			CONCAT(' Istposition: ',TO_STRING(IQ_stAchse.fPosIstwert)));
	END_IF
	
	IQ_stUniAnstgHMI.stAchsMeldHMI.bMeldEndlNeg				:= IQ_stAchse.stMeldg.bEndlNegAngf
																				OR bTestMeldAchs;

